KUKA KRL program: MyProgram_170().src

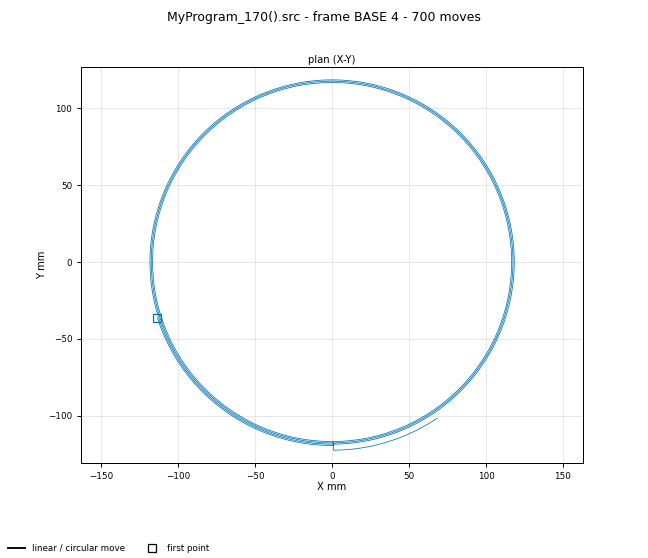
[picture p0: tool path of MyProgram_170().src in frame BASE 4, 700 of 700 moves have a stored position in this frame; points joined in program order, loops and branches not executed]
&ACCESS RVP
&REL 1
&PARAM TEMPLATE = C:\KRC\Roboter\Template\vorgabe
&PARAM EDITMASK = *
DEF MyProgram_170()
; ---- Setting reference (Base) ----
$BASE = BASE_DATA[4]

; --------------------------
; ---- Setting tool (TCP) ----
$TOOL = TOOL_DATA[3]
; --------------------------

$VEL.CP = VEL_APROX_PRINT
Startdeposition()
$VEL.CP = VEL_PRINT
LIN {X -113.5052,Y -36.4878,Z 127,A -165.8208,B 24.953,C -1.584,E1 24.8476,E2 251.9445} C_DIS
LIN {X -111.6101,Y -41.9286,Z 127,A -162.9942,B 24.9533,C -1.5781,E1 24.8503,E2 249.1159} C_DIS
LIN {X -110.2084,Y -45.4881,Z 127,A -160.9601,B 24.9532,C -1.581,E1 24.8524,E2 247.0636} C_DIS
LIN {X -109.0453,Y -48.2102,Z 127,A -158.8474,B 24.9516,C -1.6066,E1 24.8548,E2 244.8784} C_DIS
LIN {X -107.1025,Y -52.385,Z 127,A -157.3487,B 24.9538,C -1.5695,E1 24.8566,E2 243.4599} C_DIS
LIN {X -103.3826,Y -59.3866,Z 127,A -153.4546,B 24.9543,C -1.5625,E1 24.8617,E2 239.5618} C_DIS
LIN {X -101.5052,Y -62.5457,Z 127,A -151.5823,B 24.9543,C -1.5623,E1 24.8644,E2 237.6803} C_DIS
LIN {X -97.3693,Y -68.8059,Z 127,A -148.1509,B 24.9553,C -1.5454,E1 24.8698,E2 234.2721} C_DIS
LIN {X -94.1478,Y -73.1515,Z 127,A -145.4763,B 24.9554,C -1.5422,E1 24.8742,E2 231.5924} C_DIS
LIN {X -92.5246,Y -75.1928,Z 127,A -144.1286,B 24.9554,C -1.5433,E1 24.8766,E2 230.2358} C_DIS
LIN {X -89.3989,Y -78.8856,Z 127,A -141.8633,B 24.9558,C -1.5352,E1 24.8807,E2 227.9793} C_DIS
LIN {X -86.3504,Y -82.2124,Z 127,A -139.6412,B 24.956,C -1.5327,E1 24.8849,E2 225.7535} C_DIS
LIN {X -83.6012,Y -85.0038,Z 127,A -137.7658,B 24.9562,C -1.5283,E1 24.8886,E2 223.8806} C_DIS
LIN {X -80.6485,Y -87.8098,Z 127,A -135.7312,B 24.9562,C -1.5277,E1 24.8928,E2 221.8392} C_DIS
LIN {X -77.6053,Y -90.5113,Z 127,A -133.107,B 24.9548,C -1.5534,E1 24.8985,E2 219.1436} C_DIS
LIN {X -73.8299,Y -93.6156,Z 127,A -131.4433,B 24.9568,C -1.5186,E1 24.902,E2 217.5564} C_DIS
LIN {X -68.2201,Y -97.7793,Z 127,A -128.3574,B 24.9578,C -1.5007,E1 24.9088,E2 214.5022} C_DIS
LIN {X -64.8921,Y -100.0204,Z 127,A -125.9526,B 24.9568,C -1.5187,E1 24.9145,E2 212.0467} C_DIS
LIN {X -61.1405,Y -102.3566,Z 127,A -123.8263,B 24.957,C -1.5156,E1 24.9196,E2 209.9212} C_DIS
LIN {X -57.6877,Y -104.3413,Z 127,A -122.1447,B 24.9577,C -1.5025,E1 24.9236,E2 208.2656} C_DIS
LIN {X -54.8991,Y -105.8359,Z 127,A -120.1219,B 24.9565,C -1.5231,E1 24.9288,E2 206.1886} C_DIS
LIN {X -51.6513,Y -107.4564,Z 127,A -118.853,B 24.9579,C -1.4996,E1 24.9319,E2 204.9722} C_DIS
LIN {X -48.5945,Y -108.8737,Z 127,A -117.0256,B 24.9574,C -1.5071,E1 24.9366,E2 203.1225} C_DIS
LIN {X -45.5532,Y -110.1819,Z 127,A -115.4322,B 24.9575,C -1.5055,E1 24.9407,E2 201.5292} C_DIS
LIN {X -41.5744,Y -111.7442,Z 127,A -113.4125,B 24.9577,C -1.502,E1 24.9459,E2 199.5136} C_DIS
LIN {X -34.6444,Y -114.0832,Z 127,A -110.078,B 24.9584,C -1.4909,E1 24.9547,E2 196.1992} C_DIS
LIN {X -30.9247,Y -115.1452,Z 127,A -108.1569,B 24.9583,C -1.4926,E1 24.9599,E2 194.2713} C_DIS
LIN {X -27.2973,Y -116.0595,Z 127,A -106.2943,B 24.9582,C -1.4945,E1 24.965,E2 192.4014} C_DIS
LIN {X -24.0689,Y -116.7708,Z 127,A -104.8317,B 24.9585,C -1.4881,E1 24.9689,E2 190.9523} C_DIS
LIN {X -21.1691,Y -117.3312,Z 127,A -103.1394,B 24.9578,C -1.5001,E1 24.9737,E2 189.2299} C_DIS
LIN {X -17.3006,Y -117.9648,Z 127,A -100.9429,B 24.9571,C -1.514,E1 24.9798,E2 186.9985} C_DIS
LIN {X -13.2009,Y -118.4943,Z 127,A -99.5336,B 24.9586,C -1.487,E1 24.9836,E2 185.6522} C_DIS
LIN {X -9.7391,Y -118.8273,Z 127,A -97.5553,B 24.9578,C -1.5011,E1 24.9892,E2 183.6395} C_DIS
LIN {X -5.1976,Y -119.1122,Z 127,A -95.0814,B 24.957,C -1.5146,E1 24.9962,E2 181.1329} C_DIS
LIN {X -1.0081,Y -119.2216,Z 127,A -93.8519,B 24.959,C -1.4785,E1 24.9994,E2 179.989} C_DIS
LIN {X 0.8196,Y -119.2186,Z 127,A -93.0673,B 24.9593,C -1.4745,E1 25.0015,E2 179.2139} C_DIS
Enddeposition()
LIN {X 0.8196,Y -119.2186,Z 127,A -93.0673,B 24.9593,C -1.4745,E1 25.0015,E2 179.2139} C_DIS
Startdeposition()
$VEL.CP = VEL_PRINT
LIN {X -0.0391,Y -118.372,Z 127,A -93.8876,B 24.9595,C -1.4708,E1 24.9992,E2 180.043} C_DIS
LIN {X -4.3772,Y -118.2906,Z 127,A -96.2471,B 24.9601,C -1.4588,E1 24.9925,E2 182.4313} C_DIS
LIN {X -9.4244,Y -117.9943,Z 127,A -98.4039,B 24.9594,C -1.4719,E1 24.9866,E2 184.5578} C_DIS
LIN {X -12.5177,Y -117.7065,Z 127,A -99.909,B 24.9594,C -1.4719,E1 24.9824,E2 186.0636} C_DIS
LIN {X -16.6207,Y -117.1974,Z 127,A -101.8484,B 24.9592,C -1.4751,E1 24.9771,E2 187.997} C_DIS
LIN {X -20.2002,Y -116.6357,Z 127,A -103.6512,B 24.9593,C -1.4734,E1 24.9721,E2 189.8054} C_DIS
LIN {X -24.0976,Y -115.8916,Z 127,A -105.637,B 24.9594,C -1.4713,E1 24.9666,E2 191.7985} C_DIS
LIN {X -27.8137,Y -115.0562,Z 127,A -107.5207,B 24.9594,C -1.4704,E1 24.9615,E2 193.6866} C_DIS
LIN {X -31.4579,Y -114.115,Z 127,A -109.3751,B 24.9595,C -1.4701,E1 24.9565,E2 195.5447} C_DIS
LIN {X -37.8506,Y -112.1552,Z 127,A -112.5951,B 24.9593,C -1.4733,E1 24.9479,E2 198.7627} C_DIS
LIN {X -41.3491,Y -110.9148,Z 127,A -114.6072,B 24.9598,C -1.4654,E1 24.9426,E2 200.7976} C_DIS
LIN {X -45.5282,Y -109.2652,Z 127,A -116.6703,B 24.9594,C -1.4725,E1 24.9373,E2 202.8484} C_DIS
LIN {X -48.8236,Y -107.8321,Z 127,A -118.3095,B 24.959,C -1.4789,E1 24.9331,E2 204.4765} C_DIS
LIN {X -53.245,Y -105.719,Z 127,A -120.8876,B 24.9594,C -1.4728,E1 24.9266,E2 207.0757} C_DIS
LIN {X -57.5895,Y -103.4163,Z 127,A -123.0415,B 24.9586,C -1.4859,E1 24.9214,E2 209.2047} C_DIS
LIN {X -60.5891,Y -101.6887,Z 127,A -124.6802,B 24.9584,C -1.4899,E1 24.9174,E2 210.8388} C_DIS
LIN {X -64.0241,Y -99.561,Z 127,A -126.7311,B 24.9584,C -1.4888,E1 24.9125,E2 212.8988} C_DIS
LIN {X -67.4388,Y -97.2805,Z 127,A -129.3777,B 24.9599,C -1.4638,E1 24.9063,E2 215.6137} C_DIS
LIN {X -71.413,Y -94.4024,Z 127,A -131.0247,B 24.9579,C -1.4992,E1 24.9028,E2 217.1825} C_DIS
LIN {X -76.3979,Y -90.416,Z 127,A -134.0037,B 24.9573,C -1.5097,E1 24.8964,E2 220.1477} C_DIS
LIN {X -79.5446,Y -87.6616,Z 127,A -136.6302,B 24.9585,C -1.488,E1 24.8908,E2 222.8362} C_DIS
LIN {X -82.1301,Y -85.2415,Z 127,A -138.0501,B 24.9576,C -1.5041,E1 24.8879,E2 224.2236} C_DIS
LIN {X -85.6045,Y -81.7535,Z 127,A -140.7471,B 24.9581,C -1.496,E1 24.8826,E2 226.9515} C_DIS
LIN {X -88.0479,Y -79.1144,Z 127,A -142.3136,B 24.9574,C -1.5073,E1 24.8797,E2 228.4981} C_DIS
LIN {X -90.4361,Y -76.3744,Z 127,A -143.9401,B 24.9569,C -1.517,E1 24.8768,E2 230.1089} C_DIS
LIN {X -92.8607,Y -73.4055,Z 127,A -146.0087,B 24.9571,C -1.5125,E1 24.8732,E2 232.1978} C_DIS
LIN {X -95.3281,Y -70.172,Z 127,A -147.7423,B 24.9563,C -1.5273,E1 24.8703,E2 233.9047} C_DIS
LIN {X -97.4574,Y -67.1844,Z 127,A -150.0141,B 24.9572,C -1.511,E1 24.8666,E2 236.2263} C_DIS
LIN {X -99.7647,Y -63.7068,Z 127,A -151.4276,B 24.9555,C -1.5417,E1 24.8646,E2 237.574} C_DIS
LIN {X -101.44,Y -61.0057,Z 127,A -153.133,B 24.9556,C -1.5388,E1 24.8621,E2 239.295} C_DIS
LIN {X -105.283,Y -54.1019,Z 127,A -156.6636,B 24.9543,C -1.5617,E1 24.8574,E2 242.7898} C_DIS
LIN {X -108.0747,Y -48.2854,Z 127,A -159.968,B 24.9543,C -1.5629,E1 24.8534,E2 246.1091} C_DIS
LIN {X -109.1675,Y -45.7599,Z 127,A -161.341,B 24.9541,C -1.5651,E1 24.8519,E2 247.4846} C_DIS
LIN {X -110.511,Y -42.4153,Z 127,A -163.3389,B 24.9544,C -1.5597,E1 24.8499,E2 249.5065} C_DIS
LIN {X -111.9074,Y -38.5826,Z 127,A -165.0622,B 24.9535,C -1.5761,E1 24.8483,E2 251.2006} C_DIS
LIN {X -112.8699,Y -35.6687,Z 127,A -167.026,B 24.9544,C -1.5608,E1 24.8466,E2 253.2121} C_DIS
LIN {X -113.8659,Y -32.3424,Z 127,A -168.6935,B 24.954,C -1.5665,E1 24.8453,E2 254.8756} C_DIS
LIN {X -114.7916,Y -28.8912,Z 127,A -170.2491,B 24.9533,C -1.579,E1 24.8442,E2 256.4104} C_DIS
LIN {X -115.6196,Y -25.3692,Z 127,A -172.1413,B 24.9533,C -1.5787,E1 24.8431,E2 258.3144} C_DIS
LIN {X -116.2672,Y -22.2132,Z 127,A -173.7179,B 24.953,C -1.583,E1 24.8423,E2 259.8903} C_DIS
LIN {X -116.8505,Y -18.9152,Z 127,A -175.0809,B 24.9521,C -1.5987,E1 24.8417,E2 261.2238} C_DIS
LIN {X -117.3768,Y -15.3026,Z 127,A -176.7695,B 24.9516,C -1.6077,E1 24.841,E2 262.9012} C_DIS
LIN {X -117.7742,Y -11.8707,Z 127,A -178.5046,B 24.9514,C -1.6104,E1 24.8405,E2 264.6401} C_DIS
LIN {X -118.0959,Y -8.0522,Z 127,A 179.6712,B 24.951,C -1.6177,E1 24.8401,E2 266.4579} C_DIS
LIN {X -118.273,Y -4.8014,Z 127,A 177.9752,B 24.951,C -1.6179,E1 24.8399,E2 268.1637} C_DIS
LIN {X -118.3676,Y -0.795,Z 127,A 176.1264,B 24.9503,C -1.6279,E1 24.8398,E2 269.9997} C_DIS
LIN {X -118.3344,Y 2.9784,Z 127,A 174.167,B 24.9503,C -1.6284,E1 24.8398,E2 271.9697} C_DIS
LIN {X -118.1771,Y 6.7602,Z 127,A 172.4742,B 24.9496,C -1.6402,E1 24.8401,E2 273.6447} C_DIS
LIN {X -117.9183,Y 10.345,Z 127,A 170.6106,B 24.9496,C -1.6407,E1 24.8405,E2 275.5181} C_DIS
LIN {X -117.5437,Y 13.9637,Z 127,A 168.9118,B 24.949,C -1.6491,E1 24.841,E2 277.2073} C_DIS
LIN {X -117.011,Y 17.8867,Z 127,A 167.0072,B 24.9486,C -1.6558,E1 24.8418,E2 279.1072} C_DIS
LIN {X -116.4927,Y 20.9982,Z 127,A 165.4577,B 24.9484,C -1.6598,E1 24.8425,E2 280.6562} C_DIS
LIN {X -115.8224,Y 24.4345,Z 127,A 163.6134,B 24.9484,C -1.6591,E1 24.8436,E2 282.5131} C_DIS
LIN {X -114.6859,Y 29.3025,Z 127,A 161.3054,B 24.9476,C -1.6715,E1 24.8451,E2 284.805} C_DIS
LIN {X -113.8896,Y 32.2588,Z 127,A 159.8566,B 24.9473,C -1.6776,E1 24.8461,E2 286.2478} C_DIS
LIN {X -113.0444,Y 35.1059,Z 127,A 158.409,B 24.947,C -1.6818,E1 24.8473,E2 287.6937} C_DIS
LIN {X -112.1631,Y 37.8273,Z 127,A 156.3231,B 24.9485,C -1.6574,E1 24.8493,E2 289.8496} C_DIS
LIN {X -110.5995,Y 42.1817,Z 127,A 154.7269,B 24.9464,C -1.6908,E1 24.8507,E2 291.3754} C_DIS
LIN {X -109.1675,Y 45.7599,Z 127,A 152.7887,B 24.9463,C -1.6935,E1 24.8528,E2 293.3177} C_DIS
LIN {X -107.3603,Y 49.8522,Z 127,A 150.6937,B 24.9456,C -1.7031,E1 24.8552,E2 295.4015} C_DIS
LIN {X -105.9876,Y 52.7079,Z 127,A 149.1524,B 24.9454,C -1.7074,E1 24.8571,E2 296.9409} C_DIS
LIN {X -103.2744,Y 57.8436,Z 127,A 146.4293,B 24.9446,C -1.7194,E1 24.8606,E2 299.6498} C_DIS
LIN {X -102.0009,Y 60.061,Z 127,A 144.7359,B 24.9456,C -1.7042,E1 24.8631,E2 301.3882} C_DIS
LIN {X -99.5565,Y 64.0312,Z 127,A 142.7748,B 24.9444,C -1.7228,E1 24.8659,E2 303.3149} C_DIS
LIN {X -97.0332,Y 67.7946,Z 127,A 140.5953,B 24.9439,C -1.7296,E1 24.8694,E2 305.4891} C_DIS
LIN {X -95.1489,Y 70.4167,Z 127,A 138.7223,B 24.9445,C -1.721,E1 24.8725,E2 307.3917} C_DIS
LIN {X -92.2509,Y 74.1717,Z 127,A 136.197,B 24.9447,C -1.7177,E1 24.8769,E2 309.9367} C_DIS
LIN {X -89.771,Y 77.1551,Z 127,A 134.73,B 24.9433,C -1.7396,E1 24.8795,E2 311.3582} C_DIS
LIN {X -86.16,Y 81.1661,Z 127,A 132.229,B 24.9425,C -1.7509,E1 24.8842,E2 313.8433} C_DIS
LIN {X -84.1818,Y 83.2159,Z 127,A 130.2291,B 24.944,C -1.7284,E1 24.8882,E2 315.9052} C_DIS
LIN {X -81.1968,Y 86.1311,Z 127,A 128.8246,B 24.942,C -1.7589,E1 24.8909,E2 317.243} C_DIS
LIN {X -77.3367,Y 89.6158,Z 127,A 126.2723,B 24.9417,C -1.7632,E1 24.8962,E2 319.7952} C_DIS
LIN {X -75.1375,Y 91.4673,Z 127,A 124.5657,B 24.9424,C -1.7531,E1 24.9,E2 321.5324} C_DIS
LIN {X -72.2059,Y 93.7964,Z 127,A 123.031,B 24.9414,C -1.7687,E1 24.9033,E2 323.0356} C_DIS
LIN {X -69.3987,Y 95.8943,Z 127,A 120.7851,B 24.9427,C -1.7491,E1 24.9085,E2 325.3359} C_DIS
LIN {X -66.2082,Y 98.1223,Z 127,A 119.3893,B 24.9411,C -1.7734,E1 24.9116,E2 326.6786} C_DIS
LIN {X -61.9954,Y 100.8382,Z 127,A 116.5115,B 24.942,C -1.759,E1 24.9185,E2 329.5999} C_DIS
LIN {X -58.8396,Y 102.7102,Z 127,A 115.3406,B 24.9401,C -1.7878,E1 24.9211,E2 330.7057} C_DIS
LIN {X -56.4035,Y 104.0678,Z 127,A 113.8298,B 24.9404,C -1.7833,E1 24.9249,E2 332.2315} C_DIS
LIN {X -50.0829,Y 107.2529,Z 127,A 110.6953,B 24.9392,C -1.8013,E1 24.9326,E2 335.3314} C_DIS
LIN {X -46.7025,Y 108.7694,Z 127,A 108.4739,B 24.9402,C -1.7856,E1 24.9384,E2 337.5955} C_DIS
LIN {X -37.5657,Y 112.2513,Z 127,A 103.7704,B 24.9397,C -1.7931,E1 24.9507,E2 342.2909} C_DIS
LIN {X -30.0285,Y 114.4993,Z 127,A 100.0754,B 24.9391,C -1.8021,E1 24.9606,E2 345.9706} C_DIS
LIN {X -26.7678,Y 115.3038,Z 127,A 98.3933,B 24.9391,C -1.8012,E1 24.9651,E2 347.6571} C_DIS
LIN {X -23.2649,Y 116.0626,Z 127,A 96.5392,B 24.9394,C -1.7975,E1 24.9702,E2 349.5222} C_DIS
LIN {X -19.524,Y 116.7488,Z 127,A 94.7867,B 24.9391,C -1.8028,E1 24.975,E2 351.264} C_DIS
LIN {X -15.8816,Y 117.3018,Z 127,A 92.9793,B 24.9391,C -1.8028,E1 24.98,E2 353.0727} C_DIS
LIN {X -11.5481,Y 117.8065,Z 127,A 90.9936,B 24.9386,C -1.8096,E1 24.9855,E2 355.0437} C_DIS
LIN {X -7.3764,Y 118.1416,Z 127,A 88.9639,B 24.9386,C -1.8103,E1 24.9911,E2 357.0725} C_DIS
LIN {X -4.7319,Y 118.2759,Z 127,A 87.6215,B 24.9387,C -1.808,E1 24.9949,E2 358.4204} C_DIS
LIN {X -1.0943,Y 118.3656,Z 127,A 85.7256,B 24.9391,C -1.8025,E1 25.0002,E2 360.3296} C_DIS
LIN {X 3.5309,Y 118.3174,Z 127,A 83.8582,B 24.938,C -1.8193,E1 25.0053,E2 362.1569} C_DIS
LIN {X 6.4272,Y 118.1955,Z 127,A 82.1561,B 24.9389,C -1.8061,E1 25.0102,E2 363.8899} C_DIS
LIN {X 9.5709,Y 117.9826,Z 127,A 80.6683,B 24.9388,C -1.8077,E1 25.0143,E2 365.3732} C_DIS
LIN {X 13.5439,Y 117.5929,Z 127,A 79.0111,B 24.9379,C -1.8197,E1 25.0188,E2 367.0007} C_DIS
LIN {X 16.0243,Y 117.2821,Z 127,A 77.4073,B 24.9392,C -1.8018,E1 25.0234,E2 368.6457} C_DIS
LIN {X 19.694,Y 116.7204,Z 127,A 75.7682,B 24.9387,C -1.8083,E1 25.0278,E2 370.2678} C_DIS
LIN {X 22.6023,Y 116.1923,Z 127,A 74.3871,B 24.9386,C -1.8099,E1 25.0316,E2 371.6434} C_DIS
LIN {X 25.4423,Y 115.6037,Z 127,A 72.9371,B 24.9388,C -1.8072,E1 25.0356,E2 373.0981} C_DIS
LIN {X 28.3955,Y 114.9143,Z 127,A 71.3558,B 24.9392,C -1.8012,E1 25.0399,E2 374.6912} C_DIS
LIN {X 34.8507,Y 113.1236,Z 127,A 68.1216,B 24.9393,C -1.7993,E1 25.0486,E2 377.9245} C_DIS
LIN {X 38.5303,Y 111.9257,Z 127,A 66.0495,B 24.94,C -1.7886,E1 25.0541,E2 380.0179} C_DIS
LIN {X 42.7614,Y 110.3777,Z 127,A 63.9893,B 24.9398,C -1.792,E1 25.0595,E2 382.0656} C_DIS
LIN {X 45.9227,Y 109.0989,Z 127,A 62.5568,B 24.9393,C -1.8002,E1 25.0631,E2 383.4754} C_DIS
LIN {X 48.8106,Y 107.838,Z 127,A 61.0315,B 24.9393,C -1.7985,E1 25.067,E2 385.0011} C_DIS
LIN {X 52.0995,Y 106.2892,Z 127,A 59.1406,B 24.9399,C -1.7903,E1 25.0718,E2 386.9064} C_DIS
LIN {X 55.3131,Y 104.6516,Z 127,A 57.4712,B 24.9399,C -1.7915,E1 25.0759,E2 388.5684} C_DIS
LIN {X 58.2116,Y 103.0689,Z 127,A 55.9486,B 24.9398,C -1.7927,E1 25.0796,E2 390.0836} C_DIS
LIN {X 61.7564,Y 100.9838,Z 127,A 53.7966,B 24.9405,C -1.7823,E1 25.0848,E2 392.2536} C_DIS
LIN {X 67.3124,Y 97.3684,Z 127,A 50.6083,B 24.9408,C -1.7779,E1 25.0923,E2 395.4415} C_DIS
LIN {X 70.1982,Y 95.3089,Z 127,A 48.915,B 24.9408,C -1.776,E1 25.0961,E2 397.1335} C_DIS
LIN {X 73.4299,Y 92.8414,Z 127,A 47.2388,B 24.9402,C -1.786,E1 25.0997,E2 398.78} C_DIS
LIN {X 75.615,Y 91.0705,Z 127,A 45.6807,B 24.941,C -1.7742,E1 25.1031,E2 400.36} C_DIS
LIN {X 78.4344,Y 88.6556,Z 127,A 43.9958,B 24.9409,C -1.7758,E1 25.1067,E2 402.0344} C_DIS
LIN {X 80.872,Y 86.4365,Z 127,A 42.283,B 24.9415,C -1.767,E1 25.1102,E2 403.7609} C_DIS
LIN {X 83.2605,Y 84.1378,Z 127,A 40.7076,B 24.9416,C -1.765,E1 25.1133,E2 405.3346} C_DIS
LIN {X 85.4293,Y 81.9353,Z 127,A 39.1605,B 24.942,C -1.7593,E1 25.1164,E2 406.8885} C_DIS
LIN {X 88.1254,Y 79.0278,Z 127,A 37.3203,B 24.942,C -1.7587,E1 25.1198,E2 408.7221} C_DIS
LIN {X 90.5606,Y 76.2282,Z 127,A 35.0099,B 24.9439,C -1.7302,E1 25.1241,E2 411.089} C_DIS
LIN {X 93.0544,Y 73.1604,Z 127,A 33.6326,B 24.9425,C -1.7508,E1 25.1264,E2 412.4113} C_DIS
LIN {X 94.8055,Y 70.8764,Z 127,A 32.1828,B 24.943,C -1.7447,E1 25.1288,E2 413.8687} C_DIS
LIN {X 97.1116,Y 67.6817,Z 127,A 30.322,B 24.9431,C -1.742,E1 25.1319,E2 415.7267} C_DIS
LIN {X 98.9873,Y 64.9081,Z 127,A 28.6756,B 24.9435,C -1.7366,E1 25.1344,E2 417.3778} C_DIS
LIN {X 101.3152,Y 61.2111,Z 127,A 26.6858,B 24.9435,C -1.7369,E1 25.1373,E2 419.3568} C_DIS
LIN {X 103.0363,Y 58.2701,Z 127,A 24.814,B 24.9444,C -1.7218,E1 25.14,E2 421.2546} C_DIS
LIN {X 104.7359,Y 55.153,Z 127,A 23.3231,B 24.944,C -1.7278,E1 25.1419,E2 422.7233} C_DIS
LIN {X 106.2159,Y 52.2472,Z 127,A 21.7683,B 24.9443,C -1.7245,E1 25.1438,E2 424.2777} C_DIS
LIN {X 107.3966,Y 49.7742,Z 127,A 20.4355,B 24.9445,C -1.7204,E1 25.1454,E2 425.6129} C_DIS
LIN {X 108.8474,Y 46.5195,Z 127,A 18.4811,B 24.9456,C -1.7044,E1 25.1476,E2 427.5944} C_DIS
LIN {X 111.4418,Y 39.9084,Z 127,A 15.3105,B 24.9454,C -1.7069,E1 25.1508,E2 430.7415} C_DIS
LIN {X 112.6377,Y 36.3897,Z 127,A 13.1631,B 24.9468,C -1.6848,E1 25.1527,E2 432.9288} C_DIS
LIN {X 113.9399,Y 32.0813,Z 127,A 11.3534,B 24.9461,C -1.6958,E1 25.1541,E2 434.7024} C_DIS
LIN {X 114.8577,Y 28.6272,Z 127,A 9.4765,B 24.9469,C -1.6833,E1 25.1554,E2 436.5978} C_DIS
LIN {X 115.6861,Y 25.0645,Z 127,A 7.8329,B 24.9469,C -1.6838,E1 25.1564,E2 438.2306} C_DIS
LIN {X 116.4159,Y 21.4252,Z 127,A 5.9819,B 24.9474,C -1.6755,E1 25.1574,E2 440.0904} C_DIS
LIN {X 116.9915,Y 18.0131,Z 127,A 4.382,B 24.9474,C -1.6738,E1 25.1581,E2 441.6849} C_DIS
LIN {X 117.5642,Y 13.7887,Z 127,A 2.6172,B 24.947,C -1.6816,E1 25.1587,E2 443.4209} C_DIS
LIN {X 117.8265,Y 11.3395,Z 127,A 1.0957,B 24.9483,C -1.6618,E1 25.1592,E2 444.9801} C_DIS
LIN {X 118.1045,Y 7.9251,Z 127,A -0.6235,B 24.9488,C -1.6535,E1 25.1595,E2 446.7086} C_DIS
LIN {X 118.3273,Y 3.2081,Z 127,A -2.7355,B 24.9488,C -1.6544,E1 25.1598,E2 448.8059} C_DIS
LIN {X 118.3719,Y 0.1148,Z 127,A -4.3724,B 24.9494,C -1.6428,E1 25.1598,E2 450.4605} C_DIS
LIN {X 118.3222,Y -3.3749,Z 127,A -6.2151,B 24.9502,C -1.6299,E1 25.1597,E2 452.3227} C_DIS
LIN {X 118.1098,Y -7.8461,Z 127,A -8.3069,B 24.9504,C -1.6264,E1 25.1593,E2 454.4103} C_DIS
LIN {X 117.7254,Y -12.3368,Z 127,A -10.2372,B 24.9501,C -1.6314,E1 25.1588,E2 456.3174} C_DIS
LIN {X 117.3174,Y -15.7608,Z 127,A -11.8659,B 24.9503,C -1.6278,E1 25.1582,E2 457.9448} C_DIS
LIN {X 116.4381,Y -21.3016,Z 127,A -14.5672,B 24.9508,C -1.6197,E1 25.157,E2 460.6495} C_DIS
LIN {X 115.756,Y -24.7439,Z 127,A -16.7756,B 24.9527,C -1.5896,E1 25.1557,E2 462.916} C_DIS
LIN {X 114.8884,Y -28.4982,Z 127,A -18.5325,B 24.9527,C -1.5888,E1 25.1545,E2 464.6646} C_DIS
LIN {X 113.9941,Y -31.8899,Z 127,A -19.8617,B 24.952,C -1.601,E1 25.1536,E2 465.9573} C_DIS
LIN {X 113.0382,Y -35.1262,Z 127,A -21.4503,B 24.9522,C -1.598,E1 25.1523,E2 467.5439} C_DIS
LIN {X 111.8313,Y -38.7995,Z 127,A -23.3565,B 24.9526,C -1.5904,E1 25.1506,E2 469.4573} C_DIS
LIN {X 110.5817,Y -42.2287,Z 127,A -25.0488,B 24.9527,C -1.5884,E1 25.149,E2 471.1448} C_DIS
LIN {X 109.541,Y -44.8587,Z 127,A -26.7135,B 24.9538,C -1.5699,E1 25.1472,E2 472.8439} C_DIS
LIN {X 106.5024,Y -51.6606,Z 127,A -30.017,B 24.9536,C -1.5734,E1 25.1434,E2 476.1213} C_DIS
LIN {X 105.2235,Y -54.2184,Z 127,A -31.5278,B 24.9542,C -1.5632,E1 25.1414,E2 477.6483} C_DIS
LIN {X 102.927,Y -58.4623,Z 127,A -33.5975,B 24.9539,C -1.569,E1 25.1387,E2 479.6934} C_DIS
LIN {X 101.1507,Y -61.4817,Z 127,A -35.6022,B 24.955,C -1.5492,E1 25.1357,E2 481.7344} C_DIS
LIN {X 98.6653,Y -65.3965,Z 127,A -37.8368,B 24.9554,C -1.5432,E1 25.1323,E2 483.972} C_DIS
LIN {X 96.1082,Y -69.1004,Z 127,A -39.9563,B 24.9556,C -1.5399,E1 25.1289,E2 486.0889} C_DIS
LIN {X 93.858,Y -72.1261,Z 127,A -41.5271,B 24.9552,C -1.5471,E1 25.1263,E2 487.6353} C_DIS
LIN {X 91.9925,Y -74.4907,Z 127,A -43.0605,B 24.9556,C -1.5396,E1 25.1236,E2 489.1793} C_DIS
LIN {X 90.0245,Y -76.8575,Z 127,A -44.7955,B 24.9565,C -1.5239,E1 25.1204,E2 490.9433} C_DIS
LIN {X 86.0412,Y -81.2924,Z 127,A -47.4854,B 24.9564,C -1.5259,E1 25.1154,E2 493.6168} C_DIS
LIN {X 83.2368,Y -84.1612,Z 127,A -49.3,B 24.9564,C -1.5271,E1 25.1118,E2 495.4207} C_DIS
LIN {X 79.7155,Y -87.5048,Z 127,A -51.8883,B 24.9573,C -1.5101,E1 25.1065,E2 498.0385} C_DIS
LIN {X 76.266,Y -90.5284,Z 127,A -54.0133,B 24.9573,C -1.5095,E1 25.102,E2 500.1567} C_DIS
LIN {X 71.506,Y -94.3315,Z 127,A -56.8477,B 24.9573,C -1.5085,E1 25.0958,E2 502.983} C_DIS
LIN {X 68.7382,Y -96.3666,Z 127,A -58.4961,B 24.9575,C -1.5057,E1 25.0921,E2 504.6322} C_DIS
LIN {X 65.6173,Y -98.5197,Z 127,A -60.3469,B 24.9578,C -1.5012,E1 25.0878,E2 506.4874} C_DIS
LIN {X 61.2981,Y -101.2623,Z 127,A -62.6636,B 24.9576,C -1.504,E1 25.0824,E2 508.7901} C_DIS
LIN {X 57.2915,Y -103.5821,Z 127,A -65.3512,B 24.959,C -1.4789,E1 25.0757,E2 511.5289} C_DIS
LIN {X 54.3392,Y -105.1618,Z 127,A -66.479,B 24.9579,C -1.4992,E1 25.073,E2 512.6056} C_DIS
LIN {X 49.8797,Y -107.3475,Z 127,A -68.948,B 24.9583,C -1.4923,E1 25.0668,E2 515.0846} C_DIS
LIN {X 47.2005,Y -108.5523,Z 127,A -70.4294,B 24.9586,C -1.4873,E1 25.063,E2 516.574} C_DIS
LIN {X 44.1599,Y -109.8254,Z 127,A -71.9393,B 24.9585,C -1.489,E1 25.0591,E2 518.0766} C_DIS
LIN {X 41.5941,Y -110.822,Z 127,A -73.3192,B 24.9587,C -1.4849,E1 25.0555,E2 519.4631} C_DIS
LIN {X 38.7174,Y -111.8601,Z 127,A -75.4265,B 24.9604,C -1.454,E1 25.0498,E2 521.6393} C_DIS
LIN {X 34.4596,Y -113.2448,Z 127,A -76.9183,B 24.9588,C -1.4825,E1 25.046,E2 523.0608} C_DIS
LIN {X 31.4936,Y -114.1054,Z 127,A -78.5825,B 24.9594,C -1.473,E1 25.0414,E2 524.7447} C_DIS
LIN {X 27.8038,Y -115.0586,Z 127,A -80.2693,B 24.9591,C -1.4785,E1 25.0369,E2 526.4161} C_DIS
LIN {X 24.9338,Y -115.7146,Z 127,A -81.6804,B 24.9591,C -1.4778,E1 25.0331,E2 527.827} C_DIS
LIN {X 21.814,Y -116.3441,Z 127,A -83.9521,B 24.961,C -1.443,E1 25.0266,E2 530.1784} C_DIS
LIN {X 17.1261,Y -117.1256,Z 127,A -85.6737,B 24.9596,C -1.4677,E1 25.022,E2 531.84} C_DIS
LIN {X 13.557,Y -117.5913,Z 127,A -87.3639,B 24.9596,C -1.469,E1 25.0174,E2 533.5257} C_DIS
LIN {X 8.2486,Y -118.0826,Z 127,A -89.8445,B 24.9594,C -1.4722,E1 25.0105,E2 535.9973} C_DIS
LIN {X 3.6002,Y -118.3153,Z 127,A -91.7618,B 24.9586,C -1.4867,E1 25.0052,E2 537.8797} C_DIS
LIN {X 0.8127,Y -118.3652,Z 127,A -93.0641,B 24.9585,C -1.4885,E1 25.0016,E2 539.1776} C_DIS
Enddeposition()
LIN {X 0.8127,Y -118.3652,Z 127,A -93.0641,B 24.9585,C -1.4885,E1 25.0016,E2 539.1776} C_DIS
Startdeposition()
$VEL.CP = VEL_PRINT
LIN {X 2.1297,Y -117.4953,Z 127,A -92.0846,B 24.9568,C -1.519,E1 25.0045,E2 538.126} C_DIS
LIN {X 5.3393,Y -117.3936,Z 127,A -90.6038,B 24.957,C -1.5156,E1 25.0086,E2 536.6535} C_DIS
LIN {X 9.1957,Y -117.1543,Z 127,A -88.6092,B 24.9566,C -1.5216,E1 25.0142,E2 534.6457} C_DIS
LIN {X 12.8768,Y -116.8087,Z 127,A -86.7221,B 24.9563,C -1.5265,E1 25.0195,E2 532.7483} C_DIS
LIN {X 17.1396,Y -116.2596,Z 127,A -84.6573,B 24.9563,C -1.5265,E1 25.0252,E2 530.6853} C_DIS
LIN {X 21.8235,Y -115.4711,Z 127,A -82.4681,B 24.9566,C -1.5225,E1 25.0312,E2 528.5079} C_DIS
LIN {X 24.549,Y -114.9229,Z 127,A -81.24,B 24.9568,C -1.5178,E1 25.0345,E2 527.2924} C_DIS
LIN {X 27.9366,Y -114.1456,Z 127,A -79.361,B 24.9563,C -1.528,E1 25.0397,E2 525.3919} C_DIS
LIN {X 31.8574,Y -113.1142,Z 127,A -77.4736,B 24.9563,C -1.526,E1 25.0448,E2 523.5123} C_DIS
LIN {X 36.3357,Y -111.756,Z 127,A -75.1577,B 24.9561,C -1.5303,E1 25.0509,E2 521.1904} C_DIS
LIN {X 39.4625,Y -110.692,Z 127,A -73.4554,B 24.9558,C -1.5367,E1 25.0555,E2 519.4765} C_DIS
LIN {X 42.5556,Y -109.5394,Z 127,A -72.0297,B 24.9561,C -1.5303,E1 25.0591,E2 518.0689} C_DIS
LIN {X 45.7524,Y -108.2423,Z 127,A -70.2431,B 24.9557,C -1.5377,E1 25.0638,E2 516.269} C_DIS
LIN {X 48.9669,Y -106.8288,Z 127,A -68.4673,B 24.9554,C -1.5433,E1 25.0683,E2 514.4843} C_DIS
LIN {X 52.9182,Y -104.9273,Z 127,A -66.5654,B 24.9558,C -1.5357,E1 25.073,E2 512.6054} C_DIS
LIN {X 55.0014,Y -103.8489,Z 127,A -64.4009,B 24.9528,C -1.5863,E1 25.0787,E2 510.3275} C_DIS
LIN {X 60.1988,Y -100.9257,Z 127,A -62.3613,B 24.955,C -1.5502,E1 25.0833,E2 508.3795} C_DIS
LIN {X 63.3483,Y -98.9782,Z 127,A -60.7765,B 24.9554,C -1.5432,E1 25.087,E2 506.8163} C_DIS
LIN {X 65.3937,Y -97.6406,Z 127,A -59.5594,B 24.9552,C -1.5468,E1 25.0899,E2 505.5947} C_DIS
LIN {X 67.1788,Y -96.4194,Z 127,A -58.2832,B 24.9544,C -1.5595,E1 25.0929,E2 504.2928} C_DIS
LIN {X 69.7592,Y -94.5701,Z 127,A -56.0258,B 24.9522,C -1.5969,E1 25.0981,E2 501.9553} C_DIS
LIN {X 74.0846,Y -91.2204,Z 127,A -54.2272,B 24.9543,C -1.561,E1 25.1018,E2 500.2482} C_DIS
LIN {X 77.0633,Y -88.7187,Z 127,A -52.3115,B 24.954,C -1.5663,E1 25.1059,E2 498.3275} C_DIS
LIN {X 79.2932,Y -86.7312,Z 127,A -50.8024,B 24.9537,C -1.5723,E1 25.109,E2 496.8104} C_DIS
LIN {X 82.3423,Y -83.8423,Z 127,A -48.8305,B 24.9537,C -1.5736,E1 25.113,E2 494.8435} C_DIS
LIN {X 84.6789,Y -81.4811,Z 127,A -47.1847,B 24.9533,C -1.5789,E1 25.1162,E2 493.1923} C_DIS
LIN {X 87.5462,Y -78.3922,Z 127,A -45.0836,B 24.9528,C -1.5864,E1 25.1202,E2 491.0827} C_DIS
LIN {X 90.2345,Y -75.2825,Z 127,A -43.1621,B 24.9528,C -1.5877,E1 25.1236,E2 489.1669} C_DIS
LIN {X 92.7135,Y -72.2098,Z 127,A -41.2012,B 24.9524,C -1.5946,E1 25.1271,E2 487.1989} C_DIS
LIN {X 95.0734,Y -69.0718,Z 127,A -38.6614,B 24.9502,C -1.6304,E1 25.1314,E2 484.587} C_DIS
LIN {X 97.8757,Y -65.04,Z 127,A -37.089,B 24.9522,C -1.5972,E1 25.1337,E2 483.1007} C_DIS
LIN {X 99.1487,Y -63.0828,Z 127,A -35.7316,B 24.9514,C -1.6111,E1 25.1358,E2 481.7174} C_DIS
LIN {X 100.9663,Y -60.1302,Z 127,A -34.3738,B 24.952,C -1.5999,E1 25.1377,E2 480.3929} C_DIS
LIN {X 102.5635,Y -57.3621,Z 127,A -32.0782,B 24.9496,C -1.6404,E1 25.1409,E2 478.0137} C_DIS
LIN {X 104.5503,Y -53.6559,Z 127,A -29.9951,B 24.9491,C -1.6481,E1 25.1436,E2 475.9234} C_DIS
LIN {X 106.4862,Y -49.703,Z 127,A -27.9963,B 24.9491,C -1.6475,E1 25.1459,E2 473.9368} C_DIS
LIN {X 108.069,Y -46.1638,Z 127,A -26.4407,B 24.9498,C -1.6369,E1 25.1476,E2 472.4146} C_DIS
LIN {X 109.5428,Y -42.5471,Z 127,A -24.5517,B 24.9495,C -1.6422,E1 25.1496,E2 470.5238} C_DIS
LIN {X 110.7729,Y -39.2321,Z 127,A -23.1414,B 24.9501,C -1.6324,E1 25.1509,E2 469.1445} C_DIS
LIN {X 111.6405,Y -36.6928,Z 127,A -21.5013,B 24.9488,C -1.6526,E1 25.1524,E2 467.466} C_DIS
LIN {X 112.705,Y -33.2759,Z 127,A -20.0211,B 24.9493,C -1.6453,E1 25.1535,E2 466.0113} C_DIS
LIN {X 114.9212,Y -24.5568,Z 127,A -15.5751,B 24.9482,C -1.6622,E1 25.1566,E2 461.5512} C_DIS
LIN {X 115.5077,Y -21.6335,Z 127,A -14.2121,B 24.9482,C -1.6625,E1 25.1572,E2 460.1954} C_DIS
LIN {X 116.045,Y -18.5354,Z 127,A -12.7313,B 24.9481,C -1.665,E1 25.1579,E2 458.7175} C_DIS
LIN {X 116.5295,Y -15.1841,Z 127,A -11.125,B 24.9478,C -1.6682,E1 25.1586,E2 457.1131} C_DIS
LIN {X 117.0095,Y -10.8836,Z 127,A -8.9542,B 24.9472,C -1.6781,E1 25.1592,E2 454.9319} C_DIS
LIN {X 117.2976,Y -7.1695,Z 127,A -7.1501,B 24.9469,C -1.6834,E1 25.1595,E2 453.126} C_DIS
LIN {X 117.4396,Y -4.2456,Z 127,A -5.5656,B 24.9461,C -1.6958,E1 25.1597,E2 451.5217} C_DIS
LIN {X 117.5113,Y -0.9207,Z 127,A -4.0807,B 24.9461,C -1.6944,E1 25.1597,E2 450.0488} C_DIS
LIN {X 117.4927,Y 2.2687,Z 127,A -2.4519,B 24.9456,C -1.7031,E1 25.1597,E2 448.4093} C_DIS
LIN {X 117.3771,Y 5.722,Z 127,A -0.6774,B 24.945,C -1.7129,E1 25.1595,E2 446.6222} C_DIS
LIN {X 117.083,Y 10.0875,Z 127,A 1.2275,B 24.9453,C -1.7087,E1 25.1591,E2 444.7384} C_DIS
LIN {X 116.738,Y 13.4888,Z 127,A 2.8258,B 24.9451,C -1.7108,E1 25.1586,E2 443.1446} C_DIS
LIN {X 116.3731,Y 16.3401,Z 127,A 4.3289,B 24.9445,C -1.7203,E1 25.1581,E2 441.6282} C_DIS
LIN {X 115.8907,Y 19.4683,Z 127,A 5.783,B 24.9445,C -1.7209,E1 25.1574,E2 440.1811} C_DIS
LIN {X 115.4498,Y 21.9339,Z 127,A 6.9293,B 24.9445,C -1.7211,E1 25.1568,E2 439.041} C_DIS
LIN {X 114.8044,Y 25.0923,Z 127,A 8.6434,B 24.9437,C -1.733,E1 25.1559,E2 437.3089} C_DIS
LIN {X 113.8955,Y 28.941,Z 127,A 10.5196,B 24.9435,C -1.7365,E1 25.1546,E2 435.4354} C_DIS
LIN {X 113.1663,Y 31.6733,Z 127,A 11.719,B 24.9438,C -1.7321,E1 25.1537,E2 434.2531} C_DIS
LIN {X 112.6,Y 33.6296,Z 127,A 13.3945,B 24.9414,C -1.7682,E1 25.1523,E2 432.502} C_DIS
LIN {X 111.4203,Y 37.3529,Z 127,A 14.7814,B 24.9427,C -1.7489,E1 25.1512,E2 431.1685} C_DIS
LIN {X 110.5478,Y 39.8627,Z 127,A 16.6421,B 24.9406,C -1.7801,E1 25.1494,E2 429.2446} C_DIS
LIN {X 109.0388,Y 43.8232,Z 127,A 18.2414,B 24.9417,C -1.7636,E1 25.1477,E2 427.6931} C_DIS
LIN {X 107.6341,Y 47.1659,Z 127,A 19.9504,B 24.9416,C -1.7659,E1 25.1459,E2 425.988} C_DIS
LIN {X 106.1943,Y 50.3273,Z 127,A 21.7,B 24.9411,C -1.7735,E1 25.1438,E2 424.2301} C_DIS
LIN {X 104.3279,Y 54.091,Z 127,A 23.6591,B 24.941,C -1.775,E1 25.1413,E2 422.2778} C_DIS
LIN {X 102.9219,Y 56.7202,Z 127,A 25.1964,B 24.9404,C -1.783,E1 25.1392,E2 420.7297} C_DIS
LIN {X 100.8279,Y 60.3642,Z 127,A 27.2672,B 24.94,C -1.7896,E1 25.1363,E2 418.654} C_DIS
LIN {X 99.0377,Y 63.2556,Z 127,A 28.6088,B 24.9407,C -1.7789,E1 25.1344,E2 417.3444} C_DIS
LIN {X 97.7318,Y 65.2582,Z 127,A 29.8536,B 24.9402,C -1.7857,E1 25.1324,E2 416.0898} C_DIS
LIN {X 95.8389,Y 68.0049,Z 127,A 31.7727,B 24.939,C -1.8038,E1 25.1293,E2 414.1372} C_DIS
LIN {X 93.1794,Y 71.6051,Z 127,A 34.4493,B 24.937,C -1.8329,E1 25.1247,E2 411.4046} C_DIS
LIN {X 89.913,Y 75.6692,Z 127,A 36.3579,B 24.9387,C -1.8086,E1 25.1214,E2 409.5622} C_DIS
LIN {X 87.5835,Y 78.3505,Z 127,A 37.9312,B 24.9389,C -1.8052,E1 25.1185,E2 408.0041} C_DIS
LIN {X 84.9979,Y 81.1501,Z 127,A 40.0686,B 24.9377,C -1.8225,E1 25.1143,E2 405.8351} C_DIS
LIN {X 81.3944,Y 84.7625,Z 127,A 42.3301,B 24.9381,C -1.8172,E1 25.1099,E2 403.5956} C_DIS
LIN {X 78.8359,Y 87.1483,Z 127,A 44.2524,B 24.9372,C -1.8309,E1 25.1059,E2 401.6488} C_DIS
LIN {X 75.1884,Y 90.3127,Z 127,A 46.3441,B 24.9377,C -1.8231,E1 25.1015,E2 399.5835} C_DIS
LIN {X 72.0474,Y 92.8386,Z 127,A 48.6119,B 24.9365,C -1.841,E1 25.0964,E2 397.2819} C_DIS
LIN {X 68.2562,Y 95.6596,Z 127,A 51.5777,B 24.934,C -1.8762,E1 25.0895,E2 394.2431} C_DIS
LIN {X 63.0124,Y 99.1938,Z 127,A 53.5964,B 24.9371,C -1.8311,E1 25.085,E2 392.3376} C_DIS
LIN {X 59.9608,Y 101.0663,Z 127,A 55.1796,B 24.9375,C -1.8263,E1 25.0813,E2 390.7708} C_DIS
LIN {X 57.235,Y 102.6344,Z 127,A 56.9456,B 24.9366,C -1.8393,E1 25.0769,E2 388.9795} C_DIS
LIN {X 53.6984,Y 104.5285,Z 127,A 58.8855,B 24.9365,C -1.8411,E1 25.0721,E2 387.0405} C_DIS
LIN {X 50.1093,Y 106.297,Z 127,A 60.8223,B 24.9363,C -1.8429,E1 25.0673,E2 385.1047} C_DIS
LIN {X 47.5388,Y 107.4715,Z 127,A 62.2813,B 24.936,C -1.8482,E1 25.0635,E2 383.6367} C_DIS
LIN {X 44.0693,Y 108.9387,Z 127,A 64.0052,B 24.9362,C -1.845,E1 25.0591,E2 381.9244} C_DIS
LIN {X 40.3094,Y 110.3849,Z 127,A 65.7596,B 24.9367,C -1.8373,E1 25.0546,E2 380.1919} C_DIS
LIN {X 36.8547,Y 111.5881,Z 127,A 67.8296,B 24.9357,C -1.8519,E1 25.049,E2 378.0915} C_DIS
LIN {X 29.3227,Y 113.7974,Z 127,A 71.5629,B 24.9358,C -1.8503,E1 25.0391,E2 374.3682} C_DIS
LIN {X 26.0318,Y 114.5958,Z 127,A 73.3402,B 24.9354,C -1.8569,E1 25.0342,E2 372.5778} C_DIS
LIN {X 22.4685,Y 115.3469,Z 127,A 74.8568,B 24.9361,C -1.846,E1 25.0301,E2 371.0888} C_DIS
LIN {X 20.0007,Y 115.8017,Z 127,A 76.3427,B 24.9353,C -1.8583,E1 25.0259,E2 369.5755} C_DIS
LIN {X 16.254,Y 116.3854,Z 127,A 78.1391,B 24.9353,C -1.8565,E1 25.021,E2 367.785} C_DIS
LIN {X 12.1337,Y 116.8865,Z 127,A 79.972,B 24.936,C -1.8483,E1 25.016,E2 365.9728} C_DIS
LIN {X 9.712,Y 117.1131,Z 127,A 81.2638,B 24.9356,C -1.8531,E1 25.0123,E2 364.6703} C_DIS
LIN {X 6.373,Y 117.3417,Z 127,A 82.7901,B 24.936,C -1.8484,E1 25.0081,E2 363.1558} C_DIS
LIN {X 2.9606,Y 117.479,Z 127,A 84.5158,B 24.9358,C -1.8509,E1 25.0033,E2 361.4245} C_DIS
LIN {X 0.4933,Y 117.5137,Z 127,A 85.8668,B 24.9353,C -1.8573,E1 24.9995,E2 360.0584} C_DIS
LIN {X -2.9659,Y 117.4789,Z 127,A 87.3789,B 24.9359,C -1.8491,E1 24.9953,E2 358.5656} C_DIS
LIN {X -6.3369,Y 117.3437,Z 127,A 88.9647,B 24.9361,C -1.846,E1 24.9909,E2 356.987} C_DIS
LIN {X -8.7465,Y 117.1902,Z 127,A 90.2923,B 24.9357,C -1.8521,E1 24.9872,E2 355.6444} C_DIS
LIN {X -12.1987,Y 116.8797,Z 127,A 92.0688,B 24.9355,C -1.8551,E1 24.9822,E2 353.8598} C_DIS
LIN {X -15.8667,Y 116.4404,Z 127,A 93.712,B 24.9361,C -1.847,E1 24.9777,E2 352.2346} C_DIS
LIN {X -19.356,Y 115.9095,Z 127,A 95.5688,B 24.9357,C -1.8518,E1 24.9725,E2 350.3648} C_DIS
LIN {X -23.4124,Y 115.1589,Z 127,A 97.5514,B 24.9359,C -1.8489,E1 24.9671,E2 348.3869} C_DIS
LIN {X -27.2762,Y 114.3067,Z 127,A 99.3514,B 24.9364,C -1.8415,E1 24.9623,E2 346.6022} C_DIS
LIN {X -30.6399,Y 113.4498,Z 127,A 101.5466,B 24.935,C -1.8617,E1 24.9562,E2 344.3556} C_DIS
LIN {X -34.0899,Y 112.4635,Z 127,A 103.0143,B 24.936,C -1.8474,E1 24.9524,E2 342.9194} C_DIS
LIN {X -37.8269,Y 111.2604,Z 127,A 104.9176,B 24.9362,C -1.8446,E1 24.9473,E2 341.0191} C_DIS
LIN {X -44.8324,Y 108.628,Z 127,A 108.5501,B 24.9366,C -1.8389,E1 24.9379,E2 337.3925} C_DIS
LIN {X -47.589,Y 107.4496,Z 127,A 109.9002,B 24.9371,C -1.8319,E1 24.9345,E2 336.0559} C_DIS
LIN {X -50.6189,Y 106.0542,Z 127,A 111.7738,B 24.9365,C -1.84,E1 24.9297,E2 334.1582} C_DIS
LIN {X -54.6279,Y 104.0456,Z 127,A 113.7491,B 24.9374,C -1.8273,E1 24.9248,E2 332.2077} C_DIS
LIN {X -57.9428,Y 102.2389,Z 127,A 115.7253,B 24.9372,C -1.8299,E1 24.92,E2 330.2198} C_DIS
LIN {X -61.566,Y 100.0984,Z 127,A 118.1687,B 24.9363,C -1.8429,E1 24.914,E2 327.738} C_DIS
LIN {X -64.7257,Y 98.0829,Z 127,A 119.4745,B 24.9381,C -1.817,E1 24.9111,E2 326.4894} C_DIS
LIN {X -67.8117,Y 95.9768,Z 127,A 121.4412,B 24.9379,C -1.8195,E1 24.9066,E2 324.5102} C_DIS
LIN {X -70.2987,Y 94.1694,Z 127,A 122.8065,B 24.9385,C -1.8107,E1 24.9035,E2 323.161} C_DIS
LIN {X -72.6997,Y 92.328,Z 127,A 124.1243,B 24.9392,C -1.8008,E1 24.9007,E2 321.8618} C_DIS
LIN {X -75.0072,Y 90.4633,Z 127,A 125.7682,B 24.9389,C -1.806,E1 24.8971,E2 320.1994} C_DIS
LIN {X -77.0656,Y 88.7167,Z 127,A 127.2991,B 24.9385,C -1.8121,E1 24.8938,E2 318.648} C_DIS
LIN {X -80.2636,Y 85.8344,Z 127,A 129.2516,B 24.9392,C -1.8009,E1 24.8898,E2 316.7142} C_DIS
LIN {X -84.0483,Y 82.1338,Z 127,A 131.9364,B 24.9393,C -1.799,E1 24.8845,E2 314.0227} C_DIS
LIN {X -87.1725,Y 78.8096,Z 127,A 134.123,B 24.9398,C -1.7918,E1 24.8804,E2 311.8437} C_DIS
LIN {X -89.2993,Y 76.3895,Z 127,A 135.66,B 24.9402,C -1.7863,E1 24.8776,E2 310.3127} C_DIS
LIN {X -91.9315,Y 73.2015,Z 127,A 137.6566,B 24.9406,C -1.7801,E1 24.8741,E2 308.3215} C_DIS
LIN {X -93.9997,Y 70.5246,Z 127,A 139.2191,B 24.9411,C -1.772,E1 24.8714,E2 306.7708} C_DIS
LIN {X -95.3808,Y 68.647,Z 127,A 140.5587,B 24.9408,C -1.7773,E1 24.8692,E2 305.4121} C_DIS
LIN {X -99.0545,Y 63.2295,Z 127,A 143.4845,B 24.9421,C -1.7572,E1 24.8648,E2 302.5196} C_DIS
LIN {X -101.8895,Y 58.5509,Z 127,A 146.6773,B 24.9412,C -1.7714,E1 24.8601,E2 299.2765} C_DIS
LIN {X -104.4635,Y 53.8257,Z 127,A 148.8058,B 24.9431,C -1.7429,E1 24.8574,E2 297.2046} C_DIS
LIN {X -105.8987,Y 50.9424,Z 127,A 150.4676,B 24.9431,C -1.742,E1 24.8553,E2 295.536} C_DIS
LIN {X -106.8786,Y 48.8573,Z 127,A 151.6225,B 24.9433,C -1.7399,E1 24.854,E2 294.3799} C_DIS
LIN {X -108.1665,Y 45.9323,Z 127,A 153.319,B 24.9433,C -1.7408,E1 24.8521,E2 292.6718} C_DIS
LIN {X -109.6289,Y 42.3278,Z 127,A 155.1316,B 24.9438,C -1.7314,E1 24.8502,E2 290.8714} C_DIS
LIN {X -110.7907,Y 39.1812,Z 127,A 156.594,B 24.9446,C -1.7192,E1 24.8488,E2 289.4299} C_DIS
LIN {X -111.7997,Y 36.2007,Z 127,A 158.4294,B 24.9441,C -1.7268,E1 24.8472,E2 287.5659} C_DIS
LIN {X -113.0295,Y 32.156,Z 127,A 160.5409,B 24.9444,C -1.7223,E1 24.8455,E2 285.4529} C_DIS
LIN {X -114.1616,Y 27.8713,Z 127,A 162.5488,B 24.9453,C -1.709,E1 24.8442,E2 283.465} C_DIS
LIN {X -114.9693,Y 24.3359,Z 127,A 164.5344,B 24.9451,C -1.7123,E1 24.843,E2 281.4599} C_DIS
LIN {X -115.5284,Y 21.5255,Z 127,A 165.9788,B 24.9452,C -1.7097,E1 24.8422,E2 280.0131} C_DIS
LIN {X -116.1404,Y 17.9185,Z 127,A 167.5846,B 24.9461,C -1.6966,E1 24.8415,E2 278.4291} C_DIS
LIN {X -116.633,Y 14.3853,Z 127,A 169.3173,B 24.9464,C -1.6906,E1 24.8409,E2 276.7003} C_DIS
LIN {X -116.9935,Y 11.0571,Z 127,A 171.0294,B 24.9466,C -1.6886,E1 24.8404,E2 274.9826} C_DIS
LIN {X -117.2699,Y 7.5863,Z 127,A 172.8496,B 24.9466,C -1.6881,E1 24.84,E2 273.1527} C_DIS
LIN {X -117.4487,Y 3.9478,Z 127,A 174.4153,B 24.9475,C -1.6736,E1 24.8398,E2 271.6121} C_DIS
LIN {X -117.5092,Y 1.2536,Z 127,A 175.8971,B 24.9473,C -1.6763,E1 24.8398,E2 270.1151} C_DIS
LIN {X -117.4948,Y -2.1561,Z 127,A 177.5116,B 24.9478,C -1.6689,E1 24.8398,E2 268.5085} C_DIS
LIN {X -117.3896,Y -5.4318,Z 127,A 179.2338,B 24.9478,C -1.6689,E1 24.84,E2 266.776} C_DIS
LIN {X -117.1682,Y -9.0218,Z 127,A -179.212,B 24.9487,C -1.6549,E1 24.8403,E2 265.2458} C_DIS
LIN {X -116.9506,Y -11.521,Z 127,A -177.7084,B 24.9482,C -1.6625,E1 24.8407,E2 263.7148} C_DIS
LIN {X -116.5061,Y -15.3642,Z 127,A -176.1027,B 24.9493,C -1.6449,E1 24.8413,E2 262.1418} C_DIS
LIN {X -115.7525,Y -20.2806,Z 127,A -173.0282,B 24.9481,C -1.6642,E1 24.8427,E2 259.0027} C_DIS
LIN {X -114.9916,Y -24.2274,Z 127,A -171.4554,B 24.9495,C -1.6418,E1 24.8436,E2 257.4741} C_DIS
LIN {X -114.1945,Y -27.7362,Z 127,A -168.9309,B 24.9478,C -1.6688,E1 24.8453,E2 254.8706} C_DIS
LIN {X -112.7374,Y -33.1665,Z 127,A -166.9359,B 24.9503,C -1.6288,E1 24.8468,E2 252.9592} C_DIS
LIN {X -111.561,Y -36.9355,Z 127,A -164.9729,B 24.9505,C -1.6246,E1 24.8485,E2 250.9952} C_DIS
LIN {X -110.1584,Y -40.9305,Z 127,A -162.8885,B 24.9509,C -1.6192,E1 24.8504,E2 248.9117} C_DIS
LIN {X -108.8196,Y -44.3617,Z 127,A -161.1944,B 24.9514,C -1.6097,E1 24.8522,E2 247.2308} C_DIS
LIN {X -107.4496,Y -47.589,Z 127,A -159.5641,B 24.952,C -1.6014,E1 24.854,E2 245.6114} C_DIS
LIN {X -105.9055,Y -50.9283,Z 127,A -157.7447,B 24.9522,C -1.5973,E1 24.8561,E2 243.7917} C_DIS
LIN {X -104.5519,Y -53.6526,Z 127,A -156.2285,B 24.9524,C -1.5946,E1 24.8581,E2 242.274} C_DIS
LIN {X -103.1514,Y -56.2988,Z 127,A -154.3992,B 24.9517,C -1.6061,E1 24.8605,E2 240.4074} C_DIS
LIN {X -101.5237,Y -59.1871,Z 127,A -152.9798,B 24.9524,C -1.5934,E1 24.8625,E2 239.011} C_DIS
LIN {X -99.8667,Y -61.9391,Z 127,A -151.6887,B 24.9534,C -1.5776,E1 24.8643,E2 237.751} C_DIS
LIN {X -98.778,Y -63.6602,Z 127,A -150.4323,B 24.9529,C -1.5861,E1 24.8663,E2 236.4679} C_DIS
LIN {X -96.4521,Y -67.1318,Z 127,A -148.4664,B 24.9534,C -1.5779,E1 24.8693,E2 234.5119} C_DIS
LIN {X -94.1129,Y -70.374,Z 127,A -146.5821,B 24.9538,C -1.5702,E1 24.8724,E2 232.6367} C_DIS
LIN {X -91.738,Y -73.446,Z 127,A -144.4883,B 24.9536,C -1.5741,E1 24.8761,E2 230.5237} C_DIS
LIN {X -89.4642,Y -76.196,Z 127,A -142.8163,B 24.954,C -1.5672,E1 24.8791,E2 228.8605} C_DIS
LIN {X -86.7998,Y -79.2185,Z 127,A -141.1322,B 24.9549,C -1.5507,E1 24.8822,E2 227.2081} C_DIS
LIN {X -84.9533,Y -81.1963,Z 127,A -139.5236,B 24.9544,C -1.5601,E1 24.8853,E2 225.57} C_DIS
LIN {X -82.9164,Y -83.2752,Z 127,A -138.153,B 24.9547,C -1.555,E1 24.888,E2 224.2058} C_DIS
LIN {X -80.6113,Y -85.5074,Z 127,A -136.3999,B 24.9544,C -1.5599,E1 24.8916,E2 222.434} C_DIS
LIN {X -77.3822,Y -88.4403,Z 127,A -134.4135,B 24.955,C -1.5496,E1 24.8957,E2 220.4641} C_DIS
LIN {X -75.2092,Y -90.2954,Z 127,A -132.8428,B 24.9547,C -1.5546,E1 24.8991,E2 218.8755} C_DIS
LIN {X -71.6631,Y -93.1348,Z 127,A -130.7871,B 24.9554,C -1.5436,E1 24.9036,E2 216.8384} C_DIS
LIN {X -68.7642,Y -95.2972,Z 127,A -128.8215,B 24.955,C -1.5493,E1 24.908,E2 214.8523} C_DIS
LIN {X -64.9494,Y -97.9354,Z 127,A -126.9807,B 24.9563,C -1.5273,E1 24.9122,E2 213.0577} C_DIS
LIN {X -62.1551,Y -99.7318,Z 127,A -125.1544,B 24.9559,C -1.5337,E1 24.9165,E2 211.2102} C_DIS
LIN {X -58.713,Y -101.7963,Z 127,A -123.0904,B 24.9559,C -1.5356,E1 24.9215,E2 209.1356} C_DIS
LIN {X -54.9362,Y -103.8831,Z 127,A -120.3202,B 24.9543,C -1.5622,E1 24.9285,E2 206.2943} C_DIS
LIN {X -50.2779,Y -106.218,Z 127,A -118.4365,B 24.9561,C -1.5299,E1 24.9331,E2 204.4825} C_DIS
LIN {X -47.6205,Y -107.4359,Z 127,A -117.0128,B 24.9562,C -1.5283,E1 24.9367,E2 203.0593} C_DIS
LIN {X -45.0869,Y -108.5228,Z 127,A -115.8185,B 24.9567,C -1.5202,E1 24.9397,E2 201.8814} C_DIS
LIN {X -43.0127,Y -109.3599,Z 127,A -114.3967,B 24.9559,C -1.5339,E1 24.9435,E2 200.4241} C_DIS
LIN {X -38.7514,Y -110.9416,Z 127,A -112.651,B 24.9572,C -1.511,E1 24.948,E2 198.7292} C_DIS
LIN {X -32.0303,Y -113.0652,Z 127,A -109.0114,B 24.9569,C -1.5174,E1 24.9578,E2 195.0682} C_DIS
LIN {X -28.3959,Y -114.0336,Z 127,A -107.1089,B 24.9568,C -1.5193,E1 24.9629,E2 193.1583} C_DIS
LIN {X -25.1672,Y -114.7881,Z 127,A -105.7322,B 24.9574,C -1.5078,E1 24.9666,E2 191.807} C_DIS
LIN {X -22.9623,Y -115.2513,Z 127,A -104.2883,B 24.9566,C -1.5228,E1 24.9706,E2 190.3259} C_DIS
LIN {X -19.2955,Y -115.9196,Z 127,A -102.6089,B 24.9569,C -1.516,E1 24.9752,E2 188.6609} C_DIS
LIN {X -16.087,Y -116.4091,Z 127,A -100.9161,B 24.9567,C -1.5206,E1 24.9799,E2 186.9559} C_DIS
LIN {X -12.6867,Y -116.8286,Z 127,A -99.4622,B 24.9572,C -1.5106,E1 24.9839,E2 185.5248} C_DIS
LIN {X -9.2725,Y -117.1482,Z 127,A -97.6711,B 24.9569,C -1.5159,E1 24.9889,E2 183.7202} C_DIS
LIN {X -5.0096,Y -117.4077,Z 127,A -95.6678,B 24.9571,C -1.5124,E1 24.9945,E2 181.7247} C_DIS
LIN {X -2.1364,Y -117.4951,Z 127,A -94.1776,B 24.9569,C -1.5167,E1 24.9987,E2 180.2242} C_DIS
LIN {X 0.8045,Y -117.508,Z 127,A -93.0103,B 24.9576,C -1.505,E1 25.0019,E2 179.0847} C_DIS
Enddeposition()
LIN {X 0.8045,Y -117.508,Z 127,A -93.0103,B 24.9576,C -1.505,E1 25.0019,E2 179.0847} C_DIS
Startdeposition()
$VEL.CP = VEL_PRINT
LIN {X 0.1531,Y -116.6603,Z 127,A -93.8284,B 24.958,C -1.4973,E1 24.9995,E2 179.9209} C_DIS
LIN {X -2.7024,Y -116.6291,Z 127,A -95.24,B 24.958,C -1.4967,E1 24.9956,E2 181.3341} C_DIS
LIN {X -5.7403,Y -116.5198,Z 127,A -96.715,B 24.958,C -1.4973,E1 24.9915,E2 182.8079} C_DIS
LIN {X -8.437,Y -116.355,Z 127,A -98.0434,B 24.958,C -1.4973,E1 24.9878,E2 184.1369} C_DIS
LIN {X -11.1236,Y -116.1282,Z 127,A -99.3925,B 24.958,C -1.4963,E1 24.984,E2 185.4891} C_DIS
LIN {X -14.1212,Y -115.8026,Z 127,A -100.8492,B 24.958,C -1.4975,E1 24.98,E2 186.9437} C_DIS
LIN {X -17.1193,Y -115.3983,Z 127,A -102.3351,B 24.958,C -1.4978,E1 24.9759,E2 188.4301} C_DIS
LIN {X -19.4673,Y -115.0235,Z 127,A -103.5602,B 24.958,C -1.4957,E1 24.9725,E2 189.6614} C_DIS
LIN {X -22.7599,Y -114.4196,Z 127,A -105.1498,B 24.958,C -1.4987,E1 24.9681,E2 191.2456} C_DIS
LIN {X -25.4053,Y -113.8605,Z 127,A -106.486,B 24.958,C -1.499,E1 24.9645,E2 192.5828} C_DIS
LIN {X -29.2292,Y -112.9382,Z 127,A -108.4311,B 24.9579,C -1.4995,E1 24.9592,E2 194.5294} C_DIS
LIN {X -32.5608,Y -112.0248,Z 127,A -110.0808,B 24.9577,C -1.5026,E1 24.9548,E2 196.1742} C_DIS
LIN {X -35.2697,Y -111.2018,Z 127,A -111.4996,B 24.9577,C -1.5024,E1 24.951,E2 197.596} C_DIS
LIN {X -37.9649,Y -110.3109,Z 127,A -112.8954,B 24.9577,C -1.5035,E1 24.9473,E2 198.9918} C_DIS
LIN {X -40.6395,Y -109.3539,Z 127,A -114.2997,B 24.9577,C -1.5044,E1 24.9436,E2 200.397} C_DIS
LIN {X -43.1798,Y -108.3751,Z 127,A -115.6467,B 24.9576,C -1.5053,E1 24.9401,E2 201.7447} C_DIS
LIN {X -45.6932,Y -107.339,Z 127,A -116.9896,B 24.9575,C -1.5063,E1 24.9366,E2 203.0882} C_DIS
LIN {X -48.4427,Y -106.1271,Z 127,A -118.4639,B 24.9574,C -1.508,E1 24.9329,E2 204.562} C_DIS
LIN {X -51.3308,Y -104.7605,Z 127,A -120.0257,B 24.9573,C -1.5103,E1 24.929,E2 206.1225} C_DIS
LIN {X -53.7478,Y -103.5422,Z 127,A -121.3531,B 24.9572,C -1.512,E1 24.9257,E2 207.4493} C_DIS
LIN {X -55.8454,Y -102.4241,Z 127,A -122.579,B 24.9572,C -1.5111,E1 24.9226,E2 208.6808} C_DIS
LIN {X -58.7489,Y -100.7889,Z 127,A -124.1744,B 24.957,C -1.5152,E1 24.9188,E2 210.2713} C_DIS
LIN {X -61.1985,Y -99.3206,Z 127,A -125.5831,B 24.9569,C -1.517,E1 24.9154,E2 211.68} C_DIS
LIN {X -63.6178,Y -97.7887,Z 127,A -126.9944,B 24.9568,C -1.519,E1 24.9121,E2 213.0911} C_DIS
LIN {X -65.8734,Y -96.2826,Z 127,A -128.3482,B 24.9567,C -1.5203,E1 24.909,E2 214.4463} C_DIS
LIN {X -68.2293,Y -94.6279,Z 127,A -129.7602,B 24.9566,C -1.5228,E1 24.9057,E2 215.8573} C_DIS
LIN {X -71.0484,Y -92.5284,Z 127,A -131.5325,B 24.9565,C -1.524,E1 24.9018,E2 217.6332} C_DIS
LIN {X -73.3854,Y -90.6859,Z 127,A -132.9727,B 24.9563,C -1.5276,E1 24.8987,E2 219.0701} C_DIS
LIN {X -75.5989,Y -88.849,Z 127,A -134.387,B 24.9561,C -1.5302,E1 24.8956,E2 220.4836} C_DIS
LIN {X -77.7538,Y -86.9695,Z 127,A -135.8013,B 24.956,C -1.5326,E1 24.8927,E2 221.8977} C_DIS
LIN {X -79.8704,Y -85.0297,Z 127,A -137.1946,B 24.9558,C -1.5362,E1 24.8898,E2 223.2882} C_DIS
LIN {X -81.9782,Y -82.9995,Z 127,A -138.6238,B 24.9556,C -1.5396,E1 24.887,E2 224.7153} C_DIS
LIN {X -83.9543,Y -81.0001,Z 127,A -140.0437,B 24.9556,C -1.541,E1 24.8842,E2 226.138} C_DIS
LIN {X -85.9085,Y -78.9244,Z 127,A -141.4328,B 24.9553,C -1.5445,E1 24.8816,E2 227.5248} C_DIS
LIN {X -87.8117,Y -76.8014,Z 127,A -142.8612,B 24.9552,C -1.5466,E1 24.8789,E2 228.9547} C_DIS
LIN {X -89.7191,Y -74.5642,Z 127,A -144.3325,B 24.9551,C -1.5488,E1 24.8763,E2 230.4273} C_DIS
LIN {X -91.9319,Y -71.8212,Z 127,A -146.0241,B 24.9547,C -1.5546,E1 24.8733,E2 232.1132} C_DIS
LIN {X -93.6149,Y -69.6126,Z 127,A -147.4108,B 24.9546,C -1.5571,E1 24.871,E2 233.5007} C_DIS
LIN {X -95.1607,Y -67.4826,Z 127,A -148.7259,B 24.9544,C -1.5594,E1 24.8689,E2 234.8167} C_DIS
LIN {X -96.9934,Y -64.8237,Z 127,A -150.2974,B 24.9542,C -1.564,E1 24.8664,E2 236.3848} C_DIS
LIN {X -98.4788,Y -62.5426,Z 127,A -151.6427,B 24.954,C -1.5672,E1 24.8644,E2 237.7294} C_DIS
LIN {X -99.9811,Y -60.1117,Z 127,A -153.028,B 24.9537,C -1.5717,E1 24.8624,E2 239.111} C_DIS
LIN {X -101.4438,Y -57.6093,Z 127,A -154.4862,B 24.9536,C -1.5742,E1 24.8603,E2 240.571} C_DIS
LIN {X -102.6699,Y -55.3923,Z 127,A -155.7895,B 24.9536,C -1.5752,E1 24.8586,E2 241.8788} C_DIS
LIN {X -104.2041,Y -52.4534,Z 127,A -157.3763,B 24.9531,C -1.5814,E1 24.8566,E2 243.4592} C_DIS
LIN {X -105.3872,Y -50.0316,Z 127,A -158.7078,B 24.9529,C -1.5849,E1 24.8549,E2 244.7897} C_DIS
LIN {X -106.653,Y -47.2756,Z 127,A -160.2068,B 24.9527,C -1.5888,E1 24.8532,E2 246.2877} C_DIS
LIN {X -107.779,Y -44.6491,Z 127,A -161.618,B 24.9525,C -1.5925,E1 24.8517,E2 247.6976} C_DIS
LIN {X -109.301,Y -40.7794,Z 127,A -163.6745,B 24.9522,C -1.598,E1 24.8496,E2 249.7526} C_DIS
LIN {X -110.2662,Y -38.0922,Z 127,A -165.0862,B 24.9519,C -1.6019,E1 24.8483,E2 251.1632} C_DIS
LIN {X -111.1655,Y -35.3818,Z 127,A -166.4977,B 24.9517,C -1.6057,E1 24.8471,E2 252.5736} C_DIS
LIN {X -112.0632,Y -32.4282,Z 127,A -167.9943,B 24.9514,C -1.6112,E1 24.8459,E2 254.0658} C_DIS
LIN {X -112.8175,Y -29.6987,Z 127,A -169.4085,B 24.9512,C -1.6145,E1 24.8449,E2 255.4803} C_DIS
LIN {X -113.5068,Y -26.9453,Z 127,A -170.823,B 24.9509,C -1.618,E1 24.8439,E2 256.8947} C_DIS
LIN {X -114.129,Y -24.1744,Z 127,A -172.2312,B 24.9507,C -1.6219,E1 24.8431,E2 258.3021} C_DIS
LIN {X -114.6543,Y -21.541,Z 127,A -173.5589,B 24.9505,C -1.6257,E1 24.8424,E2 259.6285} C_DIS
LIN {X -115.1682,Y -18.602,Z 127,A -175.0349,B 24.9502,C -1.6299,E1 24.8417,E2 261.1032} C_DIS
LIN {X -115.5613,Y -15.9723,Z 127,A -176.3499,B 24.95,C -1.6337,E1 24.8412,E2 262.417} C_DIS
LIN {X -115.9509,Y -12.8545,Z 127,A -177.9025,B 24.9497,C -1.6383,E1 24.8407,E2 263.968} C_DIS
LIN {X -116.2168,Y -10.1638,Z 127,A -179.248,B 24.9495,C -1.6418,E1 24.8403,E2 265.3131} C_DIS
LIN {X -116.4414,Y -7.1581,Z 127,A 179.2682,B 24.9492,C -1.6465,E1 24.84,E2 266.7947} C_DIS
LIN {X -116.5751,Y -4.4584,Z 127,A 177.9635,B 24.9489,C -1.6517,E1 24.8399,E2 268.0947} C_DIS
LIN {X -116.6579,Y -0.6068,Z 127,A 175.9954,B 24.9487,C -1.6548,E1 24.8398,E2 270.0673} C_DIS
LIN {X -116.629,Y 2.7078,Z 127,A 174.3792,B 24.9483,C -1.6606,E1 24.8398,E2 271.6794} C_DIS
LIN {X -116.521,Y 5.7174,Z 127,A 172.8963,B 24.948,C -1.6653,E1 24.84,E2 273.1602} C_DIS
LIN {X -116.3564,Y 8.416,Z 127,A 171.5991,B 24.9477,C -1.6709,E1 24.8403,E2 274.4518} C_DIS
LIN {X -116.1457,Y 10.9348,Z 127,A 170.2504,B 24.9477,C -1.6706,E1 24.8406,E2 275.8093} C_DIS
LIN {X -115.8021,Y 14.1254,Z 127,A 168.7217,B 24.9473,C -1.6776,E1 24.8411,E2 277.3303} C_DIS
LIN {X -115.4585,Y 16.6963,Z 127,A 167.409,B 24.9471,C -1.6802,E1 24.8416,E2 278.6447} C_DIS
LIN {X -114.9707,Y 19.7833,Z 127,A 165.8859,B 24.9468,C -1.6857,E1 24.8423,E2 280.1638} C_DIS
LIN {X -114.4226,Y 22.7441,Z 127,A 164.4088,B 24.9464,C -1.6905,E1 24.8431,E2 281.6381} C_DIS
LIN {X -113.8538,Y 25.4362,Z 127,A 163.0292,B 24.9462,C -1.6938,E1 24.8439,E2 283.0182} C_DIS
LIN {X -113.1976,Y 28.2131,Z 127,A 161.6211,B 24.946,C -1.698,E1 24.8448,E2 284.4244} C_DIS
LIN {X -112.4733,Y 30.9744,Z 127,A 160.2121,B 24.9457,C -1.7022,E1 24.8458,E2 285.8315} C_DIS
LIN {X -111.6815,Y 33.7177,Z 127,A 158.8014,B 24.9454,C -1.7063,E1 24.8469,E2 287.2405} C_DIS
LIN {X -110.7755,Y 36.5872,Z 127,A 157.3199,B 24.9451,C -1.7109,E1 24.8482,E2 288.7197} C_DIS
LIN {X -109.847,Y 39.287,Z 127,A 155.9084,B 24.9449,C -1.7149,E1 24.8495,E2 290.1297} C_DIS
LIN {X -108.844,Y 41.9862,Z 127,A 154.4846,B 24.9446,C -1.7189,E1 24.8509,E2 291.5519} C_DIS
LIN {X -108.0416,Y 44.0039,Z 127,A 153.3905,B 24.9445,C -1.7211,E1 24.8521,E2 292.6468} C_DIS
LIN {X -106.7077,Y 47.1501,Z 127,A 151.7214,B 24.9441,C -1.7266,E1 24.8539,E2 294.312} C_DIS
LIN {X -105.4568,Y 49.8868,Z 127,A 150.2353,B 24.9439,C -1.7308,E1 24.8556,E2 295.7963} C_DIS
LIN {X -104.2724,Y 52.3156,Z 127,A 148.898,B 24.9436,C -1.7344,E1 24.8573,E2 297.1322} C_DIS
LIN {X -102.8497,Y 55.0607,Z 127,A 147.3418,B 24.9434,C -1.7374,E1 24.8593,E2 298.6896} C_DIS
LIN {X -101.4547,Y 57.5904,Z 127,A 145.9548,B 24.9431,C -1.7428,E1 24.8612,E2 300.0708} C_DIS
LIN {X -100.0398,Y 60.0152,Z 127,A 144.5636,B 24.9428,C -1.7463,E1 24.8632,E2 301.4609} C_DIS
LIN {X -98.8191,Y 62.0014,Z 127,A 143.348,B 24.9428,C -1.7468,E1 24.865,E2 302.6816} C_DIS
LIN {X -97.1035,Y 64.657,Z 127,A 141.841,B 24.9424,C -1.753,E1 24.8673,E2 304.1813} C_DIS
LIN {X -95.3791,Y 67.1764,Z 127,A 140.3322,B 24.9422,C -1.7568,E1 24.8697,E2 305.6885} C_DIS
LIN {X -93.797,Y 69.3669,Z 127,A 138.9894,B 24.942,C -1.7599,E1 24.8719,E2 307.0306} C_DIS
LIN {X -91.4348,Y 72.4503,Z 127,A 136.9976,B 24.9418,C -1.7616,E1 24.8753,E2 309.0277} C_DIS
LIN {X -89.3075,Y 75.0596,Z 127,A 135.4145,B 24.9414,C -1.7688,E1 24.8781,E2 310.601} C_DIS
LIN {X -87.3957,Y 77.2777,Z 127,A 133.968,B 24.9411,C -1.7722,E1 24.8808,E2 312.0459} C_DIS
LIN {X -85.5754,Y 79.2875,Z 127,A 132.6254,B 24.9409,C -1.7751,E1 24.8833,E2 313.3874} C_DIS
LIN {X -83.2119,Y 81.7631,Z 127,A 130.8716,B 24.9409,C -1.7763,E1 24.8867,E2 315.1459} C_DIS
LIN {X -80.9524,Y 84.0003,Z 127,A 129.37,B 24.9404,C -1.7826,E1 24.8897,E2 316.6389} C_DIS
LIN {X -78.9306,Y 85.9029,Z 127,A 127.9997,B 24.9402,C -1.7855,E1 24.8925,E2 318.0078} C_DIS
LIN {X -76.8066,Y 87.8071,Z 127,A 126.569,B 24.9402,C -1.7875,E1 24.8955,E2 319.4394} C_DIS
LIN {X -74.4487,Y 89.8151,Z 127,A 124.9926,B 24.94,C -1.7887,E1 24.8988,E2 321.0192} C_DIS
LIN {X -71.8293,Y 91.9255,Z 127,A 123.402,B 24.9396,C -1.7948,E1 24.9023,E2 322.6011} C_DIS
LIN {X -69.6202,Y 93.6092,Z 127,A 122.0249,B 24.9395,C -1.7972,E1 24.9054,E2 323.9776} C_DIS
LIN {X -67.1842,Y 95.3736,Z 127,A 120.5483,B 24.9393,C -1.8002,E1 24.9087,E2 325.452} C_DIS
LIN {X -65.0784,Y 96.8209,Z 127,A 119.3091,B 24.939,C -1.8034,E1 24.9116,E2 326.6878} C_DIS
LIN {X -62.5119,Y 98.4985,Z 127,A 117.7754,B 24.939,C -1.8051,E1 24.9152,E2 328.2222} C_DIS
LIN {X -60.0882,Y 99.9955,Z 127,A 116.3705,B 24.9388,C -1.8075,E1 24.9185,E2 329.6259} C_DIS
LIN {X -57.6265,Y 101.434,Z 127,A 114.9648,B 24.9386,C -1.8098,E1 24.9219,E2 331.0304} C_DIS
LIN {X -55.1295,Y 102.8124,Z 127,A 113.552,B 24.9385,C -1.8117,E1 24.9254,E2 332.4426} C_DIS
LIN {X -52.4627,Y 104.1993,Z 127,A 112.077,B 24.9383,C -1.8142,E1 24.929,E2 333.9156} C_DIS
LIN {X -50.0123,Y 105.3965,Z 127,A 110.7329,B 24.9382,C -1.8162,E1 24.9324,E2 335.2586} C_DIS
LIN {X -47.2756,Y 106.653,Z 127,A 109.2491,B 24.938,C -1.8182,E1 24.9362,E2 336.7411} C_DIS
LIN {X -44.6428,Y 107.7816,Z 127,A 107.8386,B 24.938,C -1.8201,E1 24.9398,E2 338.1504} C_DIS
LIN {X -41.9471,Y 108.8588,Z 127,A 106.4261,B 24.9377,C -1.8226,E1 24.9435,E2 339.5599} C_DIS
LIN {X -39.4252,Y 109.7968,Z 127,A 105.0828,B 24.9377,C -1.8234,E1 24.947,E2 340.9041} C_DIS
LIN {X -36.7359,Y 110.7255,Z 127,A 103.6817,B 24.9376,C -1.825,E1 24.9507,E2 342.3041} C_DIS
LIN {X -34.0237,Y 111.5887,Z 127,A 102.2731,B 24.9375,C -1.8261,E1 24.9545,E2 343.7124} C_DIS
LIN {X -31.2925,Y 112.385,Z 127,A 100.8683,B 24.9375,C -1.8273,E1 24.9582,E2 345.1167} C_DIS
LIN {X -28.4941,Y 113.1271,Z 127,A 99.4478,B 24.9373,C -1.8288,E1 24.9621,E2 346.5357} C_DIS
LIN {X -25.7146,Y 113.7911,Z 127,A 98.0742,B 24.9371,C -1.8314,E1 24.9658,E2 347.905} C_DIS
LIN {X -23.3497,Y 114.2985,Z 127,A 96.7924,B 24.9373,C -1.8284,E1 24.9693,E2 349.1954} C_DIS
LIN {X -20.0865,Y 114.9182,Z 127,A 95.215,B 24.9371,C -1.832,E1 24.9736,E2 350.7659} C_DIS
LIN {X -17.3149,Y 115.3681,Z 127,A 93.8398,B 24.9371,C -1.8331,E1 24.9774,E2 352.1396} C_DIS
LIN {X -14.2826,Y 115.7836,Z 127,A 92.3379,B 24.9369,C -1.8341,E1 24.9816,E2 353.6404} C_DIS
LIN {X -11.5826,Y 116.084,Z 127,A 91.0267,B 24.9369,C -1.8358,E1 24.9852,E2 354.9484} C_DIS
LIN {X -8.5694,Y 116.346,Z 127,A 89.5161,B 24.9369,C -1.8354,E1 24.9894,E2 356.4606} C_DIS
LIN {X -5.8714,Y 116.5126,Z 127,A 88.1861,B 24.9369,C -1.8358,E1 24.9931,E2 357.79} C_DIS
LIN {X -3.0163,Y 116.6214,Z 127,A 86.7753,B 24.9369,C -1.8358,E1 24.9971,E2 359.2008} C_DIS
LIN {X -0.1593,Y 116.6603,Z 127,A 85.3634,B 24.9369,C -1.8358,E1 25.001,E2 360.6128} C_DIS
LIN {X 2.7227,Y 116.6287,Z 127,A 83.9519,B 24.9369,C -1.8362,E1 25.005,E2 362.0232} C_DIS
LIN {X 5.731,Y 116.5204,Z 127,A 82.4845,B 24.9368,C -1.8367,E1 25.009,E2 363.4889} C_DIS
LIN {X 8.4291,Y 116.3555,Z 127,A 81.1558,B 24.9368,C -1.8367,E1 25.0127,E2 364.8172} C_DIS
LIN {X 11.429,Y 116.1,Z 127,A 79.6775,B 24.9368,C -1.8365,E1 25.0169,E2 366.295} C_DIS
LIN {X 14.9107,Y 115.7023,Z 127,A 77.9134,B 24.9369,C -1.8343,E1 25.0218,E2 368.063} C_DIS
LIN {X 18.3837,Y 115.2028,Z 127,A 76.2348,B 24.9369,C -1.8358,E1 25.0264,E2 369.7366} C_DIS
LIN {X 21.3513,Y 114.6907,Z 127,A 74.7567,B 24.9369,C -1.8352,E1 25.0304,E2 371.2143} C_DIS
LIN {X 24.1541,Y 114.1333,Z 127,A 73.3583,B 24.9369,C -1.8348,E1 25.0343,E2 372.612} C_DIS
LIN {X 28.2068,Y 113.1991,Z 127,A 71.2789,B 24.9371,C -1.8321,E1 25.0399,E2 374.695} C_DIS
LIN {X 31.0222,Y 112.4604,Z 127,A 69.8862,B 24.9371,C -1.8328,E1 25.0437,E2 376.0838} C_DIS
LIN {X 33.7431,Y 111.674,Z 127,A 68.4876,B 24.9371,C -1.8314,E1 25.0474,E2 377.4833} C_DIS
LIN {X 36.1684,Y 110.911,Z 127,A 67.2048,B 24.9373,C -1.8289,E1 25.0508,E2 378.7696} C_DIS
LIN {X 39.3099,Y 109.8388,Z 127,A 65.6258,B 24.9373,C -1.8297,E1 25.055,E2 380.3436} C_DIS
LIN {X 41.9867,Y 108.8438,Z 127,A 64.225,B 24.9373,C -1.8284,E1 25.0586,E2 381.7444} C_DIS
LIN {X 44.6456,Y 107.7804,Z 127,A 62.8213,B 24.9374,C -1.8271,E1 25.0623,E2 383.148} C_DIS
LIN {X 47.1353,Y 106.7142,Z 127,A 61.4943,B 24.9375,C -1.8257,E1 25.0657,E2 384.475} C_DIS
LIN {X 49.8745,Y 105.4627,Z 127,A 60.019,B 24.9376,C -1.8241,E1 25.0694,E2 385.9504} C_DIS
LIN {X 52.3047,Y 104.2778,Z 127,A 58.7258,B 24.9376,C -1.8241,E1 25.0726,E2 387.2403} C_DIS
LIN {X 54.8682,Y 102.9522,Z 127,A 57.2724,B 24.9379,C -1.8205,E1 25.0762,E2 388.698} C_DIS
LIN {X 57.5046,Y 101.504,Z 127,A 55.8096,B 24.9379,C -1.819,E1 25.0798,E2 390.1599} C_DIS
LIN {X 59.9709,Y 100.0667,Z 127,A 54.4108,B 24.9381,C -1.8171,E1 25.0832,E2 391.559} C_DIS
LIN {X 62.0223,Y 98.806,Z 127,A 53.1565,B 24.9385,C -1.812,E1 25.0862,E2 392.8213} C_DIS
LIN {X 64.7276,Y 97.0569,Z 127,A 51.656,B 24.9384,C -1.8131,E1 25.0897,E2 394.3142} C_DIS
LIN {X 67.1897,Y 95.3696,Z 127,A 50.2031,B 24.9385,C -1.8112,E1 25.093,E2 395.7667} C_DIS
LIN {X 69.3666,Y 93.7972,Z 127,A 48.8745,B 24.9387,C -1.8085,E1 25.096,E2 397.097} C_DIS
LIN {X 71.7192,Y 92.0115,Z 127,A 47.4361,B 24.9388,C -1.8064,E1 25.0992,E2 398.5351} C_DIS
LIN {X 74.0111,Y 90.1787,Z 127,A 46.0017,B 24.939,C -1.804,E1 25.1023,E2 399.9698} C_DIS
LIN {X 75.9461,Y 88.5532,Z 127,A 44.7064,B 24.9393,C -1.7991,E1 25.1051,E2 401.2717} C_DIS
LIN {X 78.7211,Y 86.0951,Z 127,A 42.917,B 24.9395,C -1.7968,E1 25.1088,E2 403.0592} C_DIS
LIN {X 80.9043,Y 84.0466,Z 127,A 41.4542,B 24.9397,C -1.7941,E1 25.1117,E2 404.5225} C_DIS
LIN {X 83.0023,Y 81.9754,Z 127,A 40.0403,B 24.9397,C -1.7925,E1 25.1145,E2 405.934} C_DIS
LIN {X 84.9621,Y 79.9424,Z 127,A 38.6769,B 24.9399,C -1.7905,E1 25.1171,E2 407.2963} C_DIS
LIN {X 86.867,Y 77.8682,Z 127,A 37.2902,B 24.9401,C -1.7872,E1 25.1197,E2 408.6846} C_DIS
LIN {X 88.7229,Y 75.7469,Z 127,A 35.8743,B 24.9404,C -1.7825,E1 25.1223,E2 410.1053} C_DIS
LIN {X 90.6031,Y 73.4876,Z 127,A 34.4615,B 24.9406,C -1.7805,E1 25.1248,E2 411.5163} C_DIS
LIN {X 92.4633,Y 71.1329,Z 127,A 32.968,B 24.9409,C -1.7759,E1 25.1274,E2 413.0135} C_DIS
LIN {X 94.4382,Y 68.4912,Z 127,A 31.3865,B 24.941,C -1.7736,E1 25.13,E2 414.5928} C_DIS
LIN {X 96.1116,Y 66.1227,Z 127,A 29.9756,B 24.9412,C -1.7706,E1 25.1323,E2 416.0039} C_DIS
LIN {X 97.787,Y 63.6203,Z 127,A 28.5115,B 24.9415,C -1.7674,E1 25.1345,E2 417.4682} C_DIS
LIN {X 99.2372,Y 61.3322,Z 127,A 27.1998,B 24.9416,C -1.7648,E1 25.1365,E2 418.7795} C_DIS
LIN {X 100.7128,Y 58.8777,Z 127,A 25.7901,B 24.9419,C -1.7608,E1 25.1385,E2 420.1913} C_DIS
LIN {X 102.1232,Y 56.3958,Z 127,A 24.3962,B 24.9421,C -1.7574,E1 25.1404,E2 421.5862} C_DIS
LIN {X 103.5577,Y 53.7182,Z 127,A 22.9148,B 24.9424,C -1.7537,E1 25.1423,E2 423.0684} C_DIS
LIN {X 104.8419,Y 51.1667,Z 127,A 21.52,B 24.9426,C -1.7501,E1 25.1441,E2 424.4642} C_DIS
LIN {X 105.9988,Y 48.7228,Z 127,A 20.1922,B 24.9428,C -1.7463,E1 25.1456,E2 425.7939} C_DIS
LIN {X 107.1012,Y 46.2475,Z 127,A 18.8518,B 24.9431,C -1.742,E1 25.1471,E2 427.1371} C_DIS
LIN {X 108.2624,Y 43.4616,Z 127,A 17.3821,B 24.9434,C -1.7382,E1 25.1487,E2 428.6076} C_DIS
LIN {X 109.3046,Y 40.7698,Z 127,A 15.9966,B 24.9436,C -1.7355,E1 25.1501,E2 429.9918} C_DIS
LIN {X 110.1977,Y 38.2874,Z 127,A 14.6885,B 24.9438,C -1.731,E1 25.1513,E2 431.303} C_DIS
LIN {X 111.159,Y 35.402,Z 127,A 13.2237,B 24.9441,C -1.7278,E1 25.1526,E2 432.7671} C_DIS
LIN {X 112.0451,Y 32.4921,Z 127,A 11.739,B 24.9443,C -1.7237,E1 25.1537,E2 434.2531} C_DIS
LIN {X 112.8074,Y 29.7379,Z 127,A 10.3448,B 24.9446,C -1.7197,E1 25.1548,E2 435.6486} C_DIS
LIN {X 113.3579,Y 27.556,Z 127,A 9.2163,B 24.9449,C -1.7152,E1 25.1555,E2 436.7812} C_DIS
LIN {X 114.1322,Y 24.1597,Z 127,A 7.5482,B 24.9451,C -1.7118,E1 25.1565,E2 438.4476} C_DIS
LIN {X 114.6606,Y 21.508,Z 127,A 6.2285,B 24.9453,C -1.708,E1 25.1572,E2 439.7686} C_DIS
LIN {X 115.1784,Y 18.5414,Z 127,A 4.7625,B 24.9456,C -1.7039,E1 25.1579,E2 441.2356} C_DIS
LIN {X 115.7849,Y 14.2721,Z 127,A 2.6573,B 24.946,C -1.6977,E1 25.1587,E2 443.3431} C_DIS
LIN {X 116.0837,Y 11.5858,Z 127,A 1.3376,B 24.9462,C -1.6938,E1 25.1591,E2 444.6641} C_DIS
LIN {X 116.3448,Y 8.5867,Z 127,A -0.131,B 24.9465,C -1.6895,E1 25.1594,E2 446.1342} C_DIS
LIN {X 116.5116,Y 5.8891,Z 127,A -1.4504,B 24.9468,C -1.6856,E1 25.1596,E2 447.4551} C_DIS
LIN {X 116.6217,Y 3.0086,Z 127,A -2.8632,B 24.947,C -1.6811,E1 25.1598,E2 448.8699} C_DIS
LIN {X 116.6555,Y -0.9696,Z 127,A -4.8365,B 24.9475,C -1.6738,E1 25.1598,E2 450.8487} C_DIS
LIN {X 116.5825,Y -4.2858,Z 127,A -6.4131,B 24.9477,C -1.6709,E1 25.1596,E2 452.4227} C_DIS
LIN {X 116.4417,Y -7.1534,Z 127,A -7.8134,B 24.9479,C -1.6668,E1 25.1594,E2 453.8245} C_DIS
LIN {X 116.2427,Y -9.8634,Z 127,A -9.1439,B 24.9482,C -1.6626,E1 25.1591,E2 455.1569} C_DIS
LIN {X 115.9503,Y -12.8596,Z 127,A -10.6067,B 24.9485,C -1.6585,E1 25.1587,E2 456.6207} C_DIS
LIN {X 115.6204,Y -15.5422,Z 127,A -11.9319,B 24.9487,C -1.6543,E1 25.1582,E2 457.9481} C_DIS
LIN {X 115.2052,Y -18.3683,Z 127,A -13.3182,B 24.949,C -1.6505,E1 25.1577,E2 459.3351} C_DIS
LIN {X 114.6901,Y -21.355,Z 127,A -14.7959,B 24.9492,C -1.6462,E1 25.1569,E2 460.8144} C_DIS
LIN {X 113.8593,Y -25.411,Z 127,A -16.9184,B 24.9499,C -1.6353,E1 25.1557,E2 462.9501} C_DIS
LIN {X 113.1544,Y -28.3879,Z 127,A -18.3335,B 24.9499,C -1.6346,E1 25.1548,E2 464.3586} C_DIS
LIN {X 112.4565,Y -31.0368,Z 127,A -19.6596,B 24.9501,C -1.6312,E1 25.1538,E2 465.6851} C_DIS
LIN {X 111.6809,Y -33.7199,Z 127,A -21.0122,B 24.9504,C -1.6278,E1 25.1527,E2 467.0381} C_DIS
LIN {X 110.7684,Y -36.6085,Z 127,A -22.4832,B 24.9506,C -1.6238,E1 25.1515,E2 468.5101} C_DIS
LIN {X 109.8387,Y -39.3102,Z 127,A -23.8772,B 24.9508,C -1.6198,E1 25.1502,E2 469.9058} C_DIS
LIN {X 108.843,Y -41.9886,Z 127,A -25.2711,B 24.9511,C -1.6159,E1 25.1488,E2 471.3012} C_DIS
LIN {X 107.7819,Y -44.6419,Z 127,A -26.6734,B 24.9513,C -1.6116,E1 25.1473,E2 472.7059} C_DIS
LIN {X 106.6675,Y -47.2424,Z 127,A -28.0466,B 24.9515,C -1.6081,E1 25.1458,E2 474.0798} C_DIS
LIN {X 105.4394,Y -49.9231,Z 127,A -29.4775,B 24.9518,C -1.6044,E1 25.1441,E2 475.5116} C_DIS
LIN {X 104.3131,Y -52.2335,Z 127,A -30.7376,B 24.952,C -1.6008,E1 25.1425,E2 476.7736} C_DIS
LIN {X 102.9677,Y -54.8387,Z 127,A -32.1776,B 24.9522,C -1.5964,E1 25.1407,E2 478.2162} C_DIS
LIN {X 101.5031,Y -57.5061,Z 127,A -33.6542,B 24.9525,C -1.5928,E1 25.1387,E2 479.6936} C_DIS
LIN {X 100.0656,Y -59.9727,Z 127,A -35.0494,B 24.9527,C -1.5891,E1 25.1367,E2 481.0906} C_DIS
LIN {X 98.5681,Y -62.4033,Z 127,A -36.4421,B 24.9529,C -1.5854,E1 25.1346,E2 482.4847} C_DIS
LIN {X 97.086,Y -64.6835,Z 127,A -37.7726,B 24.9531,C -1.5819,E1 25.1326,E2 483.8169} C_DIS
LIN {X 95.3679,Y -67.1922,Z 127,A -39.2454,B 24.9533,C -1.5786,E1 25.1302,E2 485.2902} C_DIS
LIN {X 93.8069,Y -69.3534,Z 127,A -40.5687,B 24.9536,C -1.5744,E1 25.128,E2 486.6172} C_DIS
LIN {X 92.0134,Y -71.7167,Z 127,A -42.0052,B 24.9537,C -1.5713,E1 25.1256,E2 488.054} C_DIS
LIN {X 90.1813,Y -74.008,Z 127,A -43.4378,B 24.9539,C -1.5679,E1 25.1231,E2 489.4882} C_DIS
LIN {X 88.3919,Y -76.1355,Z 127,A -44.7973,B 24.9541,C -1.5645,E1 25.1206,E2 490.8494} C_DIS
LIN {X 86.1292,Y -78.6839,Z 127,A -46.5097,B 24.9545,C -1.5584,E1 25.1174,E2 492.5685} C_DIS
LIN {X 84.0451,Y -80.9058,Z 127,A -47.9654,B 24.9546,C -1.5565,E1 25.1146,E2 494.0224} C_DIS
LIN {X 82.0387,Y -82.9397,Z 127,A -49.3614,B 24.9548,C -1.5534,E1 25.1118,E2 495.4198} C_DIS
LIN {X 79.9269,Y -84.9766,Z 127,A -50.7587,B 24.9548,C -1.552,E1 25.109,E2 496.8147} C_DIS
LIN {X 77.861,Y -86.8735,Z 127,A -52.1476,B 24.9551,C -1.5482,E1 25.1062,E2 498.2071} C_DIS
LIN {X 75.6515,Y -88.8042,Z 127,A -53.5818,B 24.9553,C -1.5452,E1 25.1031,E2 499.6427} C_DIS
LIN {X 73.3688,Y -90.6993,Z 127,A -55.1125,B 24.9557,C -1.5385,E1 25.0998,E2 501.1834} C_DIS
LIN {X 70.6663,Y -92.8229,Z 127,A -56.7115,B 24.9557,C -1.5389,E1 25.0963,E2 502.7755} C_DIS
LIN {X 68.3476,Y -94.5433,Z 127,A -58.1241,B 24.9557,C -1.5361,E1 25.0931,E2 504.1896} C_DIS
LIN {X 66.1242,Y -96.1106,Z 127,A -59.461,B 24.9559,C -1.5334,E1 25.09,E2 505.5285} C_DIS
LIN {X 63.7623,Y -97.6934,Z 127,A -60.8457,B 24.9561,C -1.5311,E1 25.0868,E2 506.9139} C_DIS
LIN {X 61.3221,Y -99.2434,Z 127,A -62.2588,B 24.9562,C -1.5287,E1 25.0834,E2 508.3282} C_DIS
LIN {X 59.2665,Y -100.483,Z 127,A -63.5504,B 24.9566,C -1.5213,E1 25.0803,E2 509.6333} C_DIS
LIN {X 56.2562,Y -102.2012,Z 127,A -65.1288,B 24.9565,C -1.5239,E1 25.0765,E2 511.2009} C_DIS
LIN {X 54.1009,Y -103.3562,Z 127,A -66.3162,B 24.9565,C -1.5225,E1 25.0736,E2 512.3883} C_DIS
LIN {X 51.1536,Y -104.8482,Z 127,A -67.9343,B 24.9567,C -1.52,E1 25.0695,E2 514.008} C_DIS
LIN {X 48.7084,Y -106.0055,Z 127,A -69.2763,B 24.9569,C -1.5172,E1 25.0661,E2 515.3529} C_DIS
LIN {X 45.9576,Y -107.2275,Z 127,A -70.7386,B 24.9569,C -1.5157,E1 25.0624,E2 516.8153} C_DIS
LIN {X 43.6853,Y -108.1713,Z 127,A -71.9825,B 24.9571,C -1.5124,E1 25.0591,E2 518.0643} C_DIS
LIN {X 40.7967,Y -109.2944,Z 127,A -73.4621,B 24.9571,C -1.5122,E1 25.0553,E2 519.5411} C_DIS
LIN {X 38.1085,Y -110.2605,Z 127,A -74.8612,B 24.9573,C -1.5105,E1 25.0516,E2 520.9413} C_DIS
LIN {X 35.398,Y -111.1603,Z 127,A -76.2586,B 24.9573,C -1.509,E1 25.0479,E2 522.3396} C_DIS
LIN {X 33.0702,Y -111.8736,Z 127,A -77.5182,B 24.9576,C -1.5048,E1 25.0445,E2 523.6071} C_DIS
LIN {X 29.7243,Y -112.8109,Z 127,A -79.1518,B 24.9575,C -1.5062,E1 25.0401,E2 525.2347} C_DIS
LIN {X 26.9524,Y -113.5051,Z 127,A -80.5547,B 24.9575,C -1.5048,E1 25.0363,E2 526.6388} C_DIS
LIN {X 24.1642,Y -114.1312,Z 127,A -81.956,B 24.9576,C -1.5036,E1 25.0325,E2 528.0411} C_DIS
LIN {X 20.0741,Y -114.9204,Z 127,A -84.0116,B 24.9578,C -1.5015,E1 25.0268,E2 530.0994} C_DIS
LIN {X 17.1491,Y -115.3937,Z 127,A -85.4511,B 24.9578,C -1.5011,E1 25.0229,E2 531.5383} C_DIS
LIN {X 14.2759,Y -115.7845,Z 127,A -86.8726,B 24.9578,C -1.5003,E1 25.0189,E2 532.9606} C_DIS
LIN {X 11.5908,Y -116.0832,Z 127,A -88.1995,B 24.9578,C -1.4996,E1 25.0152,E2 534.2884} C_DIS
LIN {X 8.5753,Y -116.3456,Z 127,A -89.6817,B 24.9579,C -1.499,E1 25.0111,E2 535.7712} C_DIS
LIN {X 5.8611,Y -116.5132,Z 127,A -91.019,B 24.9579,C -1.4984,E1 25.0074,E2 537.1095} C_DIS
LIN {X 3.0083,Y -116.6217,Z 127,A -92.4282,B 24.9579,C -1.4976,E1 25.0034,E2 538.5202} C_DIS
LIN {X 0.7992,Y -116.6564,Z 127,A -93.2239,B 24.9573,C -1.5103,E1 25.0013,E2 539.2857} C_DIS
Enddeposition()
LIN {X 0.8696,Y -122.3226,Z 128,A -92.8738,B 24.9615,C -1.4341,E1 25.0018,E2 539.1161} C_DIS
Startdeposition()
$VEL.CP = VEL_PRINT
LIN {X 3.4798,Y -122.279,Z 128,A -91.6395,B 24.9615,C -1.435,E1 25.0052,E2 537.8799} C_DIS
LIN {X 6.0025,Y -122.1831,Z 128,A -90.1044,B 24.9605,C -1.4523,E1 25.0096,E2 536.3043} C_DIS
LIN {X 9.4756,Y -121.9609,Z 128,A -88.6284,B 24.9608,C -1.4457,E1 25.0137,E2 534.8447} C_DIS
LIN {X 11.9905,Y -121.7414,Z 128,A -87.2948,B 24.9604,C -1.4536,E1 25.0174,E2 533.4932} C_DIS
LIN {X 15.4485,Y -121.3491,Z 128,A -85.8195,B 24.9608,C -1.4472,E1 25.0215,E2 532.0342} C_DIS
LIN {X 18.4219,Y -120.9334,Z 128,A -84.4152,B 24.9608,C -1.4481,E1 25.0254,E2 530.6291} C_DIS
LIN {X 21.3842,Y -120.4449,Z 128,A -83.0114,B 24.9607,C -1.449,E1 25.0292,E2 529.2244} C_DIS
LIN {X 23.8655,Y -119.9799,Z 128,A -81.6787,B 24.9602,C -1.4573,E1 25.0329,E2 527.8737} C_DIS
LIN {X 26.8028,Y -119.3581,Z 128,A -80.4274,B 24.9606,C -1.4511,E1 25.0363,E2 526.6388} C_DIS
LIN {X 29.7239,Y -118.6644,Z 128,A -78.872,B 24.9601,C -1.4598,E1 25.0406,E2 525.0652} C_DIS
LIN {X 33.0869,Y -117.7689,Z 128,A -77.398,B 24.9604,C -1.454,E1 25.0445,E2 523.6072} C_DIS
LIN {X 35.5107,Y -117.063,Z 128,A -76.0662,B 24.9599,C -1.4626,E1 25.0481,E2 522.2574} C_DIS
LIN {X 38.8257,Y -116.0035,Z 128,A -74.7933,B 24.9608,C -1.4472,E1 25.0514,E2 521.0233} C_DIS
LIN {X 41.2119,Y -115.1795,Z 128,A -73.2612,B 24.9597,C -1.4658,E1 25.0555,E2 519.4503} C_DIS
LIN {X 44.5611,Y -113.9233,Z 128,A -71.8695,B 24.9604,C -1.4543,E1 25.0591,E2 518.0889} C_DIS
LIN {X 47.2542,Y -112.833,Z 128,A -70.3865,B 24.9599,C -1.4622,E1 25.063,E2 516.5904} C_DIS
LIN {X 50.0091,Y -111.6394,Z 128,A -69.185,B 24.9604,C -1.4543,E1 25.066,E2 515.4106} C_DIS
LIN {X 52.303,Y -110.5854,Z 128,A -67.6541,B 24.9593,C -1.4734,E1 25.0699,E2 513.8387} C_DIS
LIN {X 55.0012,Y -109.2686,Z 128,A -66.2896,B 24.9593,C -1.4736,E1 25.0734,E2 512.4772} C_DIS
LIN {X 57.6662,Y -107.8859,Z 128,A -65.0037,B 24.9595,C -1.4701,E1 25.0765,E2 511.2032} C_DIS
LIN {X 60.7108,Y -106.2001,Z 128,A -63.38,B 24.9594,C -1.4728,E1 25.0805,E2 509.578} C_DIS
LIN {X 62.8904,Y -104.9264,Z 128,A -62.2022,B 24.9593,C -1.4747,E1 25.0833,E2 508.3992} C_DIS
LIN {X 65.4465,Y -103.3513,Z 128,A -60.7541,B 24.959,C -1.4795,E1 25.0867,E2 506.9444} C_DIS
LIN {X 68.3589,Y -101.4461,Z 128,A -59.1787,B 24.959,C -1.4801,E1 25.0904,E2 505.3729} C_DIS
Enddeposition()
END
